C05454=1112.944,404.001,-92.503,-176.618,11.577,149.492
C05455=1112.941,404.248,-92.543,-176.616,11.582,149.493
C05456=1112.937,404.494,-92.582,-176.614,11.587,149.494
C05457=1112.933,404.741,-92.621,-176.613,11.591,149.494
C05458=1112.930,404.988,-92.660,-176.611,11.596,149.495
C05459=1112.927,405.235,-92.699,-176.609,11.601,149.496
C05460=1112.923,405.482,-92.738,-176.606,11.605,149.496
C05461=1112.920,405.729,-92.778,-176.604,11.610,149.497
C05462=1112.916,405.976,-92.817,-176.603,11.615,149.498
C05463=1112.913,406.223,-92.856,-176.601,11.620,149.499
C05464=1112.909,406.470,-92.895,-176.599,11.625,149.500
C05465=1112.905,406.717,-92.935,-176.597,11.630,149.501
C05466=1112.902,406.964,-92.974,-176.595,11.635,149.501
C05467=1112.898,407.211,-93.013,-176.593,11.640,149.502
C05468=1112.895,407.457,-93.052,-176.592,11.645,149.503
C05469=1112.892,407.704,-93.091,-176.590,11.650,149.504
C05470=1112.888,407.951,-93.131,-176.588,11.655,149.505
C05471=1112.885,408.198,-93.170,-176.586,11.660,149.506
C05472=1112.881,408.445,-93.209,-176.584,11.665,149.507
C05473=1112.877,408.692,-93.249,-176.583,11.671,149.508
C05474=1112.874,408.939,-93.288,-176.581,11.677,149.509
C05475=1112.870,409.186,-93.327,-176.579,11.681,149.509
C05476=1112.867,409.432,-93.367,-176.577,11.687,149.510
C05477=1112.863,409.679,-93.406,-176.576,11.692,149.511
C05478=1112.860,409.926,-93.446,-176.574,11.697,149.512
C05479=1112.856,410.173,-93.485,-176.572,11.703,149.513
C05480=1112.853,410.419,-93.525,-176.570,11.708,149.514
C05481=1112.849,410.666,-93.564,-176.569,11.714,149.516
C05482=1112.845,410.913,-93.603,-176.567,11.720,149.517
C05483=1112.842,411.160,-93.643,-176.565,11.725,149.518
C05484=1112.839,411.407,-93.683,-176.564,11.731,149.519
C05485=1112.835,411.654,-93.722,-176.562,11.737,149.520
C05486=1112.832,411.900,-93.762,-176.561,11.742,149.521
C05487=1112.829,412.147,-93.801,-176.558,11.748,149.522
C05488=1112.824,412.395,-93.841,-176.557,11.754,149.523
C05489=1112.821,412.641,-93.881,-176.555,11.760,149.524
C05490=1112.817,412.888,-93.920,-176.554,11.765,149.525
C05491=1112.814,413.134,-93.960,-176.552,11.772,149.526
C05492=1112.810,413.381,-94.000,-176.551,11.777,149.528
C05493=1112.808,413.628,-94.040,-176.549,11.784,149.529
C05494=1112.805,413.875,-94.079,-176.548,11.789,149.530
C05495=1112.802,414.122,-94.119,-176.546,11.795,149.531
C05496=1112.801,414.368,-94.158,-176.544,11.802,149.533
C05497=1112.799,414.616,-94.198,-176.543,11.808,149.534
C05498=1112.800,414.863,-94.237,-176.541,11.814,149.535
C05499=1112.799,415.110,-94.277,-176.541,11.820,149.536
C05500=1112.799,415.356,-94.316,-176.539,11.826,149.537
C05501=1112.800,415.603,-94.356,-176.537,11.833,149.539
C05502=1112.802,415.814,-94.389,-176.536,11.838,149.540
C05503=1112.802,416.025,-94.422,-176.535,11.843,149.541
C05504=1112.805,416.236,-94.456,-176.534,11.849,149.542
C05505=1112.807,416.448,-94.489,-176.533,11.854,149.543
C05506=1112.810,416.659,-94.522,-176.532,11.860,149.545
C05507=1112.813,416.870,-94.555,-176.531,11.865,149.546
C05508=1112.817,417.081,-94.589,-176.529,11.871,149.547
C05509=1112.820,417.292,-94.622,-176.528,11.877,149.548
C05510=1112.401,417.292,-94.684,-176.521,11.881,149.547
C05511=1112.398,417.081,-94.652,-176.522,11.875,149.546
C05512=1112.394,416.870,-94.618,-176.523,11.870,149.545
C05513=1112.391,416.659,-94.585,-176.524,11.864,149.544
C05514=1112.388,416.448,-94.552,-176.526,11.858,149.543
C05515=1112.386,416.236,-94.519,-176.527,11.853,149.541
C05516=1112.384,416.025,-94.485,-176.528,11.847,149.540
C05517=1112.383,415.814,-94.451,-176.529,11.842,149.539
C05518=1112.381,415.602,-94.417,-176.530,11.836,149.538
C05519=1112.380,415.356,-94.378,-176.532,11.831,149.537
C05520=1112.379,415.109,-94.339,-176.533,11.824,149.535
C05521=1112.380,414.862,-94.300,-176.535,11.818,149.534
C05522=1112.381,414.615,-94.260,-176.536,11.812,149.533
C05523=1112.382,414.368,-94.221,-176.538,11.806,149.532
C05524=1112.384,414.122,-94.181,-176.539,11.799,149.531
C05525=1112.386,413.875,-94.141,-176.541,11.794,149.529
C05526=1112.388,413.628,-94.102,-176.543,11.787,149.528
C05527=1112.391,413.381,-94.062,-176.544,11.781,149.527
C05528=1112.395,413.135,-94.022,-176.546,11.776,149.526
C05529=1112.398,412.888,-93.983,-176.547,11.769,149.525
C05530=1112.401,412.641,-93.943,-176.549,11.764,149.523
C05531=1112.405,412.393,-93.903,-176.551,11.758,149.522
C05532=1112.409,412.147,-93.863,-176.552,11.752,149.521
C05533=1112.412,411.900,-93.824,-176.554,11.746,149.520
C05534=1112.416,411.653,-93.785,-176.555,11.741,149.519
C05535=1112.419,411.407,-93.745,-176.558,11.735,149.518
C05536=1112.423,411.160,-93.705,-176.559,11.729,149.517
C05537=1112.426,410.913,-93.666,-176.561,11.723,149.516
C05538=1112.430,410.667,-93.626,-176.563,11.718,149.515
C05539=1112.433,410.420,-93.587,-176.565,11.712,149.514
C05540=1112.437,410.173,-93.548,-176.566,11.707,149.513
C05541=1112.440,409.926,-93.507,-176.568,11.701,149.512
C05542=1112.443,409.679,-93.468,-176.570,11.695,149.511
C05543=1112.447,409.432,-93.429,-176.572,11.690,149.510
C05544=1112.451,409.185,-93.390,-176.573,11.685,149.509
C05545=1112.454,408.938,-93.350,-176.575,11.680,149.508
C05546=1112.458,408.691,-93.310,-176.577,11.674,149.507
C05547=1112.461,408.445,-93.271,-176.579,11.669,149.506
C05548=1112.465,408.198,-93.232,-176.581,11.663,149.505
C05549=1112.468,407.951,-93.193,-176.583,11.659,149.504
C05550=1112.472,407.704,-93.153,-176.584,11.653,149.503
C05551=1112.475,407.457,-93.113,-176.586,11.648,149.503
C05552=1112.479,407.210,-93.074,-176.588,11.642,149.502
C05553=1112.483,406.963,-93.035,-176.590,11.638,149.501
C05554=1112.486,406.716,-92.996,-176.592,11.633,149.500
C05555=1112.490,406.469,-92.956,-176.594,11.628,149.499
C05556=1112.493,406.222,-92.917,-176.596,11.623,149.499
C05557=1112.496,405.976,-92.878,-176.598,11.618,149.498
C05558=1112.500,405.729,-92.839,-176.600,11.613,149.497
C05559=1112.504,405.482,-92.800,-176.602,11.608,149.496
C05560=1112.507,405.235,-92.761,-176.604,11.603,149.495
C05561=1112.511,404.988,-92.721,-176.606,11.598,149.495
C05562=1112.514,404.741,-92.682,-176.608,11.593,149.494
C05563=1112.518,404.494,-92.643,-176.609,11.589,149.493
C05564=1112.521,404.248,-92.605,-176.612,11.585,149.492
C05565=1112.525,404.001,-92.565,-176.614,11.580,149.492
C05566=1112.529,403.754,-92.526,-176.616,11.575,149.491
C05567=1112.532,403.543,-92.493,-176.618,11.571,149.490
C05568=1112.535,403.331,-92.459,-176.619,11.568,149.490
C05569=1112.538,403.120,-92.426,-176.621,11.564,149.489
C05570=1112.540,402.908,-92.393,-176.623,11.560,149.489
C05571=1112.544,402.697,-92.360,-176.625,11.555,149.488
C05572=1112.547,402.486,-92.326,-176.627,11.552,149.488
C05573=1112.550,402.274,-92.293,-176.629,11.548,149.487
C05574=1112.553,402.063,-92.259,-176.630,11.544,149.487
C05575=1112.556,401.816,-92.221,-176.632,11.540,149.486
C05576=1112.560,401.569,-92.181,-176.634,11.536,149.485
C05577=1112.563,401.322,-92.142,-176.637,11.531,149.485
C05578=1112.567,401.075,-92.104,-176.639,11.527,149.484
C05579=1112.571,400.829,-92.065,-176.641,11.523,149.484
C05580=1112.574,400.582,-92.026,-176.643,11.518,149.483
C05581=1112.578,400.334,-91.988,-176.645,11.514,149.482
C05582=1112.581,400.087,-91.949,-176.648,11.510,149.482
C05583=1112.585,399.841,-91.910,-176.649,11.506,149.481
C05584=1112.589,399.593,-91.871,-176.652,11.502,149.481
C05585=1112.592,399.347,-91.833,-176.654,11.498,149.480
C05586=1112.596,399.100,-91.794,-176.656,11.494,149.480
C05587=1112.600,398.852,-91.755,-176.658,11.490,149.479
C05588=1112.603,398.606,-91.716,-176.661,11.486,149.479
C05589=1112.606,398.359,-91.677,-176.663,11.482,149.479
C05590=1112.611,398.112,-91.639,-176.666,11.478,149.478
C05591=1112.614,397.865,-91.600,-176.667,11.474,149.478
C05592=1112.618,397.618,-91.562,-176.669,11.471,149.477
C05593=1112.621,397.371,-91.522,-176.672,11.466,149.477
C05594=1112.624,397.123,-91.485,-176.674,11.463,149.476
C05595=1112.629,396.877,-91.446,-176.676,11.459,149.476
C05596=1112.632,396.630,-91.408,-176.679,11.455,149.476
C05597=1112.636,396.383,-91.368,-176.681,11.452,149.475
C05598=1112.639,396.136,-91.331,-176.683,11.448,149.475
C05599=1112.643,395.889,-91.292,-176.686,11.444,149.474
C05600=1112.647,395.642,-91.253,-176.688,11.440,149.474
C05601=1112.650,395.395,-91.215,-176.690,11.437,149.474
C05602=1112.654,395.148,-91.176,-176.692,11.434,149.473
C05603=1112.657,394.901,-91.138,-176.695,11.430,149.473
C05604=1112.661,394.654,-91.099,-176.698,11.426,149.473
C05605=1112.664,394.407,-91.061,-176.700,11.423,149.472
C05606=1112.669,394.160,-91.023,-176.702,11.420,149.472
C05607=1112.672,393.913,-90.984,-176.704,11.416,149.472
C05608=1112.676,393.666,-90.946,-176.707,11.413,149.472
C05609=1112.679,393.419,-90.908,-176.709,11.409,149.471
C05610=1112.683,393.172,-90.869,-176.711,11.406,149.471
C05611=1112.686,392.925,-90.831,-176.714,11.402,149.471
C05612=1112.690,392.677,-90.792,-176.717,11.399,149.470
C05613=1112.694,392.431,-90.755,-176.719,11.396,149.470
C05614=1112.698,392.184,-90.716,-176.722,11.393,149.470
C05615=1112.701,391.937,-90.678,-176.724,11.389,149.470
C05616=1112.704,391.690,-90.640,-176.726,11.386,149.470
C05617=1112.708,391.442,-90.602,-176.729,11.383,149.469
C05618=1112.712,391.195,-90.564,-176.731,11.380,149.469
C05619=1112.716,390.949,-90.525,-176.734,11.377,149.469
C05620=1112.719,390.702,-90.487,-176.736,11.373,149.469
C05621=1112.722,390.454,-90.449,-176.738,11.371,149.469
C05622=1112.727,390.207,-90.411,-176.741,11.368,149.468
C05623=1112.729,389.996,-90.378,-176.743,11.365,149.468
C05624=1112.733,389.784,-90.346,-176.745,11.363,149.468
C05625=1112.736,389.573,-90.313,-176.747,11.360,149.468
C05626=1112.739,389.361,-90.280,-176.750,11.357,149.468
C05627=1112.742,389.150,-90.248,-176.752,11.355,149.468
C05628=1112.745,388.938,-90.215,-176.754,11.353,149.468
C05629=1112.748,388.726,-90.183,-176.756,11.350,149.468
C05630=1112.751,388.516,-90.151,-176.758,11.347,149.468
C05631=1112.755,388.268,-90.112,-176.761,11.344,149.468
C05632=1112.759,388.021,-90.074,-176.763,11.342,149.467
C05633=1112.762,387.774,-90.037,-176.766,11.339,149.467
C05634=1112.766,387.527,-89.998,-176.768,11.336,149.467
C05635=1112.770,387.280,-89.960,-176.771,11.333,149.467
C05636=1112.773,387.033,-89.922,-176.773,11.331,149.467
C05637=1112.777,386.786,-89.885,-176.776,11.328,149.467
C05638=1112.781,386.539,-89.846,-176.779,11.325,149.467
C05639=1112.784,386.291,-89.808,-176.781,11.323,149.467
C05640=1112.788,386.045,-89.771,-176.784,11.320,149.467
C05641=1112.791,385.797,-89.733,-176.787,11.317,149.467
C05642=1112.795,385.551,-89.695,-176.789,11.315,149.467
C05643=1112.799,385.303,-89.657,-176.791,11.312,149.467
C05644=1112.803,385.056,-89.620,-176.794,11.309,149.467
C05645=1112.806,384.809,-89.582,-176.797,11.307,149.467
C05646=1112.810,384.562,-89.544,-176.799,11.305,149.467
C05647=1112.813,384.315,-89.506,-176.802,11.302,149.467
C05648=1112.817,384.068,-89.468,-176.805,11.300,149.467
C05649=1112.821,383.820,-89.431,-176.807,11.298,149.467
C05650=1112.825,383.574,-89.394,-176.810,11.295,149.467
C05651=1112.828,383.326,-89.356,-176.813,11.292,149.467
C05652=1112.832,383.080,-89.317,-176.816,11.290,149.467
C05653=1112.836,382.832,-89.280,-176.819,11.287,149.468
C05654=1112.840,382.585,-89.243,-176.822,11.284,149.468
C05655=1112.843,382.338,-89.205,-176.825,11.282,149.468
C05656=1112.847,382.091,-89.167,-176.828,11.279,149.468
C05657=1112.850,381.843,-89.130,-176.832,11.276,149.468
C05658=1112.854,381.597,-89.092,-176.836,11.273,149.468
C05659=1112.857,381.349,-89.054,-176.838,11.270,149.468
C05660=1112.861,381.102,-89.017,-176.842,11.268,149.468
C05661=1112.865,380.855,-88.979,-176.845,11.265,149.468
C05662=1112.869,380.608,-88.942,-176.848,11.263,149.469
C05663=1112.873,380.361,-88.905,-176.851,11.260,149.469
C05664=1112.876,380.114,-88.867,-176.854,11.258,149.469
C05665=1112.880,379.866,-88.830,-176.858,11.255,149.469
C05666=1112.883,379.619,-88.792,-176.861,11.252,149.469
C05667=1112.887,379.372,-88.755,-176.864,11.250,149.469
C05668=1112.891,379.125,-88.717,-176.867,11.247,149.469
C05669=1112.895,378.878,-88.680,-176.871,11.245,149.470
C05670=1112.899,378.631,-88.643,-176.874,11.242,149.470
C05671=1112.902,378.383,-88.605,-176.877,11.239,149.470
C05672=1112.906,378.137,-88.568,-176.880,11.237,149.470
C05673=1112.910,377.889,-88.531,-176.884,11.234,149.470
C05674=1112.913,377.642,-88.493,-176.887,11.231,149.470
C05675=1112.917,377.395,-88.456,-176.891,11.229,149.471
C05676=1112.921,377.148,-88.419,-176.894,11.226,149.471
C05677=1112.924,376.900,-88.381,-176.897,11.224,149.471
C05678=1112.929,376.653,-88.344,-176.900,11.221,149.471
C05679=1112.931,376.441,-88.312,-176.903,11.219,149.471
C05680=1112.935,376.230,-88.281,-176.906,11.217,149.472
C05681=1112.938,376.019,-88.249,-176.908,11.215,149.472
C05682=1112.941,375.807,-88.217,-176.911,11.213,149.472
C05683=1112.944,375.595,-88.186,-176.914,11.211,149.472
C05684=1112.947,375.383,-88.154,-176.917,11.209,149.472
C05685=1112.951,375.172,-88.121,-176.920,11.206,149.472
C05686=1112.954,374.960,-88.089,-176.922,11.204,149.473
C05687=1112.958,374.712,-88.053,-176.926,11.202,149.473
C05688=1112.961,374.465,-88.016,-176.929,11.199,149.473
C05689=1112.965,374.218,-87.979,-176.932,11.197,149.473
C05690=1112.969,373.970,-87.942,-176.936,11.194,149.473
C05691=1112.972,373.724,-87.905,-176.939,11.192,149.474
C05692=1112.977,373.477,-87.868,-176.942,11.190,149.474
C05693=1112.979,373.229,-87.831,-176.946,11.187,149.474
C05694=1112.983,372.982,-87.794,-176.949,11.185,149.474
C05695=1112.987,372.735,-87.757,-176.952,11.182,149.474
C05696=1112.992,372.487,-87.721,-176.955,11.180,149.475
C05697=1112.995,372.240,-87.683,-176.959,11.177,149.475
C05698=1112.998,371.993,-87.646,-176.962,11.175,149.475
C05699=1113.002,371.746,-87.609,-176.965,11.172,149.475
C05700=1113.006,371.499,-87.573,-176.969,11.170,149.475
C05701=1113.010,371.251,-87.535,-176.972,11.167,149.476
C05702=1113.013,371.004,-87.499,-176.975,11.165,149.476
C05703=1113.017,370.757,-87.462,-176.979,11.163,149.476
C05704=1113.021,370.510,-87.425,-176.982,11.160,149.476
C05705=1113.025,370.263,-87.389,-176.986,11.158,149.477
C05706=1113.028,370.015,-87.352,-176.989,11.155,149.477
C05707=1113.032,369.768,-87.315,-176.992,11.153,149.477
C05708=1113.036,369.521,-87.278,-176.995,11.150,149.477
C05709=1113.040,369.274,-87.242,-176.999,11.148,149.477
C05710=1113.044,369.026,-87.206,-177.002,11.145,149.478
C05711=1113.047,368.778,-87.169,-177.006,11.143,149.478
C05712=1113.051,368.531,-87.132,-177.009,11.141,149.478
C05713=1113.055,368.284,-87.095,-177.012,11.138,149.478
C05714=1113.058,368.037,-87.059,-177.016,11.136,149.479
C05715=1113.063,367.790,-87.022,-177.019,11.133,149.479
C05716=1113.067,367.543,-86.985,-177.022,11.131,149.479
C05717=1113.070,367.295,-86.950,-177.026,11.129,149.479
C05718=1113.074,367.047,-86.913,-177.029,11.126,149.480
C05719=1113.077,366.800,-86.876,-177.033,11.124,149.480
C05720=1113.081,366.553,-86.840,-177.036,11.121,149.480
C05721=1113.086,366.305,-86.803,-177.039,11.119,149.480
C05722=1113.089,366.059,-86.767,-177.043,11.116,149.481
C05723=1113.093,365.811,-86.730,-177.046,11.114,149.481
C05724=1113.096,365.565,-86.694,-177.049,11.112,149.481
C05725=1113.101,365.317,-86.658,-177.053,11.109,149.481
C05726=1113.104,365.069,-86.621,-177.056,11.107,149.482
C05727=1113.108,364.822,-86.584,-177.060,11.104,149.482
C05728=1113.111,364.574,-86.549,-177.063,11.102,149.482
C05729=1113.115,364.327,-86.512,-177.066,11.099,149.482
C05730=1113.119,364.080,-86.476,-177.070,11.097,149.483
C05731=1113.123,363.833,-86.440,-177.073,11.095,149.483
C05732=1113.127,363.586,-86.403,-177.077,11.092,149.483
C05733=1113.131,363.338,-86.367,-177.080,11.090,149.483
C05734=1113.134,363.091,-86.331,-177.083,11.088,149.484
C05735=1113.138,362.879,-86.300,-177.086,11.086,149.484
C05736=1113.140,362.667,-86.269,-177.089,11.084,149.484
C05737=1113.144,362.455,-86.238,-177.092,11.082,149.484
C05738=1113.147,362.243,-86.207,-177.095,11.080,149.485
C05739=1113.150,362.032,-86.177,-177.097,11.078,149.485
C05740=1113.154,361.820,-86.146,-177.100,11.075,149.485
C05741=1113.157,361.607,-86.114,-177.103,11.074,149.485
C05742=1113.159,361.396,-86.083,-177.106,11.071,149.485
C05743=1113.164,361.148,-86.047,-177.109,11.069,149.486
C05744=1113.168,360.901,-86.012,-177.113,11.067,149.486
C05745=1113.172,360.654,-85.975,-177.116,11.064,149.486
C05746=1113.175,360.406,-85.939,-177.120,11.062,149.486
C05747=1113.179,360.159,-85.903,-177.123,11.059,149.487
C05748=1113.183,359.912,-85.867,-177.126,11.057,149.487
C05749=1113.187,359.664,-85.831,-177.130,11.055,149.487
C05750=1113.190,359.417,-85.795,-177.133,11.052,149.487
C05751=1113.194,359.170,-85.759,-177.137,11.050,149.488
C05752=1113.198,358.922,-85.723,-177.140,11.047,149.488
C05753=1113.201,358.675,-85.687,-177.143,11.045,149.488
C05754=1113.205,358.427,-85.651,-177.147,11.043,149.488
C05755=1113.209,358.180,-85.616,-177.150,11.040,149.489
C05756=1113.213,357.932,-85.580,-177.154,11.038,149.489
C05757=1113.217,357.686,-85.544,-177.157,11.035,149.489
C05758=1113.221,357.438,-85.508,-177.160,11.034,149.489
C05759=1113.224,357.191,-85.473,-177.163,11.031,149.490
C05760=1113.229,356.943,-85.437,-177.167,11.029,149.490
C05761=1113.233,356.696,-85.401,-177.170,11.026,149.490
C05762=1113.236,356.449,-85.365,-177.174,11.023,149.490
C05763=1113.240,356.201,-85.329,-177.177,11.021,149.491
C05764=1113.243,355.954,-85.294,-177.180,11.018,149.491
C05765=1113.248,355.706,-85.258,-177.184,11.016,149.491
C05766=1113.251,355.458,-85.222,-177.187,11.014,149.491
C05767=1113.255,355.211,-85.187,-177.191,11.011,149.492
C05768=1113.259,354.964,-85.151,-177.194,11.009,149.492
C05769=1113.263,354.717,-85.116,-177.197,11.006,149.492
C05770=1113.267,354.469,-85.080,-177.201,11.004,149.492
C05771=1113.270,354.222,-85.045,-177.204,11.001,149.493
C05772=1113.275,353.974,-85.009,-177.207,10.999,149.493
C05773=1113.278,353.726,-84.973,-177.211,10.997,149.493
C05774=1113.282,353.479,-84.937,-177.214,10.994,149.493
C05775=1113.286,353.232,-84.902,-177.218,10.992,149.494
C05776=1113.290,352.985,-84.867,-177.221,10.989,149.494
C05777=1113.294,352.737,-84.831,-177.224,10.987,149.494
C05778=1113.297,352.490,-84.796,-177.228,10.984,149.494
C05779=1113.301,352.242,-84.760,-177.231,10.982,149.495
C05780=1113.305,351.995,-84.725,-177.234,10.980,149.495
C05781=1113.309,351.748,-84.689,-177.237,10.977,149.495
C05782=1113.313,351.500,-84.655,-177.241,10.975,149.495
C05783=1113.316,351.252,-84.619,-177.244,10.972,149.495
C05784=1113.320,351.005,-84.583,-177.247,10.970,149.496
C05785=1113.324,350.758,-84.548,-177.251,10.967,149.496
C05786=1113.328,350.510,-84.513,-177.254,10.965,149.496
C05787=1113.332,350.263,-84.477,-177.257,10.962,149.496
C05788=1113.336,350.015,-84.442,-177.261,10.960,149.497
C05789=1113.340,349.768,-84.407,-177.264,10.957,149.497
C05790=1113.344,349.520,-84.372,-177.268,10.954,149.497
C05791=1113.347,349.308,-84.342,-177.271,10.952,149.497
C05792=1113.350,349.096,-84.311,-177.273,10.951,149.498
C05793=1113.354,348.884,-84.281,-177.276,10.948,149.498
C05794=1113.357,348.672,-84.251,-177.279,10.946,149.498
C05795=1113.360,348.460,-84.221,-177.281,10.944,149.498
C05796=1113.363,348.248,-84.191,-177.284,10.942,149.498
C05797=1113.367,348.036,-84.161,-177.287,10.940,149.498
C05798=1113.370,347.824,-84.130,-177.289,10.938,149.498
C05799=1113.375,347.577,-84.096,-177.293,10.936,149.499
C05800=1113.378,347.329,-84.061,-177.296,10.933,149.499
C05801=1113.381,347.082,-84.025,-177.299,10.931,149.499
C05802=1113.386,346.834,-83.991,-177.302,10.928,149.499
C05803=1113.390,346.587,-83.955,-177.306,10.925,149.499
C05804=1113.394,346.339,-83.920,-177.309,10.923,149.500
C05805=1113.398,346.092,-83.885,-177.312,10.921,149.500
C05806=1113.402,345.844,-83.850,-177.316,10.918,149.500
C05807=1113.405,345.597,-83.815,-177.318,10.915,149.500
C05808=1113.409,345.349,-83.781,-177.321,10.914,149.500
C05809=1113.413,345.102,-83.745,-177.324,10.911,149.501
C05810=1113.417,344.854,-83.711,-177.328,10.909,149.501
C05811=1113.421,344.607,-83.675,-177.331,10.906,149.501
C05812=1113.424,344.359,-83.641,-177.334,10.904,149.501
C05813=1113.428,344.112,-83.606,-177.337,10.901,149.501
C05814=1113.433,343.864,-83.571,-177.341,10.899,149.502
C05815=1113.437,343.616,-83.536,-177.344,10.896,149.502
C05816=1113.441,343.369,-83.501,-177.347,10.894,149.502
C05817=1113.444,343.121,-83.467,-177.351,10.891,149.502
C05818=1113.448,342.873,-83.432,-177.353,10.888,149.502
C05819=1113.452,342.626,-83.397,-177.356,10.887,149.503
C05820=1113.456,342.379,-83.363,-177.359,10.884,149.503
C05821=1113.460,342.131,-83.328,-177.363,10.882,149.503
C05822=1113.464,341.884,-83.293,-177.366,10.879,149.503
C05823=1113.468,341.636,-83.258,-177.369,10.877,149.503
C05824=1113.472,341.389,-83.224,-177.372,10.874,149.504
C05825=1113.476,341.140,-83.189,-177.376,10.872,149.504
C05826=1113.480,340.894,-83.154,-177.379,10.869,149.504
C05827=1113.483,340.646,-83.120,-177.382,10.866,149.504
C05828=1113.488,340.398,-83.085,-177.385,10.864,149.504
C05829=1113.492,340.150,-83.050,-177.388,10.862,149.505
C05830=1113.495,339.903,-83.016,-177.391,10.860,149.505
C05831=1113.499,339.656,-82.981,-177.394,10.857,149.505
C05832=1113.503,339.409,-82.947,-177.397,10.855,149.505
C05833=1113.507,339.160,-82.912,-177.401,10.852,149.505
C05834=1113.511,338.913,-82.878,-177.404,10.850,149.506
C05835=1113.515,338.665,-82.843,-177.407,10.847,149.506
C05836=1113.519,338.418,-82.809,-177.410,10.844,149.506
C05837=1113.523,338.170,-82.775,-177.414,10.842,149.506
C05838=1113.527,337.923,-82.740,-177.417,10.840,149.506
C05839=1113.531,337.674,-82.705,-177.420,10.837,149.507
C05840=1113.535,337.427,-82.672,-177.423,10.835,149.507
C05841=1113.539,337.179,-82.637,-177.426,10.833,149.507
C05842=1113.543,336.932,-82.603,-177.429,10.830,149.507
C05843=1113.547,336.684,-82.568,-177.432,10.828,149.507
C05844=1113.550,336.437,-82.534,-177.435,10.825,149.507
C05845=1113.555,336.189,-82.500,-177.439,10.822,149.508
C05846=1113.558,335.942,-82.465,-177.442,10.820,149.508
C05847=1113.562,335.729,-82.436,-177.444,10.818,149.508
C05848=1113.565,335.518,-82.407,-177.448,10.816,149.508
C05849=1113.569,335.306,-82.377,-177.450,10.814,149.508
C05850=1113.572,335.093,-82.347,-177.453,10.812,149.509
C05851=1113.575,334.880,-82.319,-177.456,10.809,149.509
C05852=1113.579,334.669,-82.289,-177.458,10.807,149.509
C05853=1113.582,334.457,-82.260,-177.460,10.805,149.509
C05854=1113.585,334.245,-82.231,-177.464,10.803,149.509
C05855=1113.589,333.997,-82.196,-177.467,10.800,149.509
C05856=1113.593,333.749,-82.163,-177.470,10.798,149.509
C05857=1113.597,333.501,-82.128,-177.473,10.796,149.510
C05858=1113.601,333.254,-82.094,-177.476,10.794,149.510
C05859=1113.605,333.006,-82.060,-177.479,10.791,149.510
C05860=1113.609,332.759,-82.026,-177.482,10.788,149.510
C05861=1113.613,332.511,-81.993,-177.486,10.786,149.511
C05862=1113.616,332.264,-81.958,-177.489,10.783,149.511
C05863=1113.621,332.016,-81.924,-177.492,10.781,149.511
C05864=1113.625,331.768,-81.890,-177.495,10.778,149.511
C05865=1113.628,331.521,-81.856,-177.498,10.776,149.511
C05866=1113.633,331.273,-81.822,-177.501,10.773,149.511
C05867=1113.637,331.025,-81.788,-177.505,10.771,149.512
C05868=1113.640,330.778,-81.755,-177.507,10.769,149.512
C05869=1113.645,330.530,-81.720,-177.510,10.766,149.512
C05870=1113.648,330.282,-81.687,-177.514,10.764,149.512
C05871=1113.652,330.035,-81.653,-177.517,10.761,149.512
C05872=1113.656,329.788,-81.619,-177.520,10.758,149.512
C05873=1113.660,329.539,-81.585,-177.523,10.756,149.513
C05874=1113.664,329.292,-81.551,-177.527,10.754,149.513
C05875=1113.668,329.044,-81.518,-177.530,10.751,149.513
C05876=1113.672,328.797,-81.484,-177.533,10.748,149.513
C05877=1113.676,328.548,-81.450,-177.536,10.746,149.514
C05878=1113.680,328.301,-81.416,-177.539,10.743,149.514
C05879=1113.684,328.053,-81.383,-177.542,10.741,149.514
C05880=1113.688,327.805,-81.348,-177.545,10.739,149.514
C05881=1113.692,327.558,-81.315,-177.548,10.736,149.514
C05882=1113.696,327.310,-81.281,-177.551,10.734,149.514
C05883=1113.700,327.063,-81.248,-177.555,10.731,149.515
C05884=1113.704,326.815,-81.213,-177.558,10.729,149.515
C05885=1113.708,326.567,-81.180,-177.561,10.726,149.515
C05886=1113.712,326.319,-81.147,-177.564,10.724,149.515
C05887=1113.716,326.072,-81.113,-177.567,10.721,149.515
C05888=1113.719,325.824,-81.080,-177.570,10.718,149.515
C05889=1113.724,325.576,-81.047,-177.574,10.716,149.516
C05890=1113.728,325.329,-81.012,-177.576,10.714,149.516
C05891=1113.732,325.081,-80.979,-177.579,10.711,149.516
C05892=1113.736,324.833,-80.946,-177.583,10.709,149.516
C05893=1113.740,324.585,-80.912,-177.586,10.707,149.517
C05894=1113.744,324.338,-80.878,-177.589,10.704,149.517
C05895=1113.748,324.090,-80.845,-177.592,10.701,149.517
C05896=1113.752,323.843,-80.811,-177.596,10.699,149.517
C05897=1113.756,323.595,-80.778,-177.598,10.696,149.517
C05898=1113.759,323.347,-80.745,-177.602,10.694,149.517
C05899=1113.764,323.099,-80.712,-177.605,10.691,149.517
C05900=1113.768,322.851,-80.678,-177.608,10.688,149.518
C05901=1113.771,322.604,-80.645,-177.611,10.687,149.518
C05902=1113.776,322.356,-80.611,-177.614,10.684,149.518
C05903=1113.779,322.143,-80.582,-177.617,10.682,149.518
C05904=1113.783,321.932,-80.555,-177.619,10.680,149.518
C05905=1113.786,321.719,-80.526,-177.622,10.678,149.519
C05906=1113.789,321.507,-80.498,-177.625,10.675,149.519
C05907=1113.793,321.295,-80.468,-177.627,10.673,149.519
C05908=1113.796,321.083,-80.440,-177.630,10.671,149.519
C05909=1113.800,320.870,-80.411,-177.633,10.669,149.519
C05910=1113.803,320.658,-80.383,-177.636,10.667,149.519
C05911=1113.806,320.410,-80.350,-177.638,10.664,149.520
C05912=1113.811,320.162,-80.317,-177.642,10.662,149.520
C05913=1113.815,319.914,-80.284,-177.645,10.659,149.520
C05914=1113.819,319.666,-80.250,-177.648,10.657,149.520
C05915=1113.822,319.419,-80.218,-177.651,10.654,149.520
C05916=1113.826,319.171,-80.185,-177.654,10.651,149.520
C05917=1113.831,318.924,-80.152,-177.657,10.650,149.521
C05918=1113.835,318.676,-80.118,-177.660,10.647,149.521
C05919=1113.839,318.428,-80.085,-177.663,10.644,149.521
C05920=1113.843,318.180,-80.052,-177.667,10.642,149.521
C05921=1113.847,317.933,-80.019,-177.669,10.639,149.521
C05922=1113.850,317.685,-79.986,-177.673,10.637,149.522
C05923=1113.854,317.437,-79.953,-177.676,10.634,149.522
C05924=1113.858,317.188,-79.920,-177.679,10.632,149.522
C05925=1113.863,316.941,-79.887,-177.682,10.629,149.522
C05926=1113.867,316.693,-79.854,-177.685,10.626,149.522
C05927=1113.870,316.446,-79.822,-177.689,10.624,149.522
C05928=1113.874,316.198,-79.788,-177.691,10.622,149.523
C05929=1113.878,315.950,-79.755,-177.694,10.619,149.523
C05930=1113.883,315.702,-79.723,-177.698,10.617,149.523
C05931=1113.886,315.454,-79.690,-177.700,10.614,149.523
C05932=1113.890,315.207,-79.657,-177.704,10.612,149.523
C05933=1113.895,314.959,-79.624,-177.707,10.609,149.523
C05934=1113.899,314.711,-79.591,-177.710,10.607,149.524
C05935=1113.902,314.463,-79.559,-177.713,10.604,149.524
C05936=1113.907,314.215,-79.526,-177.716,10.601,149.524
C05937=1113.911,313.968,-79.493,-177.720,10.599,149.524
C05938=1113.914,313.720,-79.461,-177.722,10.597,149.524
C05939=1113.919,313.472,-79.428,-177.725,10.595,149.525
C05940=1113.923,313.224,-79.394,-177.729,10.592,149.525
C05941=1113.926,312.976,-79.363,-177.732,10.589,149.525
C05942=1113.931,312.728,-79.329,-177.735,10.587,149.525
C05943=1113.935,312.480,-79.297,-177.738,10.584,149.525
C05944=1113.938,312.233,-79.264,-177.741,10.582,149.526
C05945=1113.943,311.986,-79.232,-177.744,10.579,149.526
C05946=1113.948,311.737,-79.199,-177.747,10.576,149.526
C05947=1113.951,311.490,-79.167,-177.751,10.574,149.526
C05948=1113.955,311.241,-79.134,-177.754,10.571,149.526
C05949=1113.959,310.994,-79.102,-177.756,10.570,149.527
C05950=1113.963,310.746,-79.069,-177.759,10.567,149.527
C05951=1113.967,310.498,-79.036,-177.763,10.564,149.527
C05952=1113.971,310.250,-79.004,-177.765,10.562,149.527
C05953=1113.975,310.002,-78.971,-177.769,10.559,149.527
C05954=1113.979,309.754,-78.939,-177.772,10.556,149.527
C05955=1113.983,309.506,-78.906,-177.775,10.554,149.528
C05956=1113.987,309.259,-78.875,-177.778,10.552,149.528
C05957=1113.992,309.011,-78.842,-177.781,10.549,149.528
C05958=1113.996,308.763,-78.809,-177.785,10.546,149.528
C05959=1114.000,308.551,-78.782,-177.787,10.544,149.528
C05960=1114.002,308.338,-78.754,-177.789,10.542,149.528
C05961=1114.006,308.125,-78.726,-177.793,10.540,149.529
C05962=1114.009,307.914,-78.698,-177.795,10.538,149.529
C05963=1114.013,307.700,-78.671,-177.797,10.536,149.529
C05964=1114.016,307.489,-78.643,-177.801,10.533,149.529
C05965=1114.020,307.276,-78.616,-177.803,10.531,149.529
C05966=1114.024,307.063,-78.588,-177.805,10.529,149.529
C05967=1114.027,306.816,-78.555,-177.808,10.527,149.529
C05968=1114.031,306.568,-78.523,-177.811,10.524,149.530
C05969=1114.036,306.319,-78.491,-177.815,10.522,149.530
C05970=1114.039,306.071,-78.459,-177.818,10.519,149.530
C05971=1114.044,305.824,-78.426,-177.821,10.517,149.530
C05972=1114.048,305.576,-78.395,-177.824,10.514,149.530
C05973=1114.052,305.328,-78.362,-177.827,10.511,149.531
C05974=1114.056,305.080,-78.330,-177.830,10.510,149.531
C05975=1114.060,304.833,-78.299,-177.833,10.507,149.531
C05976=1114.064,304.585,-78.266,-177.836,10.505,149.531
C05977=1114.068,304.337,-78.234,-177.839,10.502,149.531
C05978=1114.072,304.089,-78.202,-177.842,10.499,149.531
C05979=1114.077,303.841,-78.170,-177.845,10.497,149.532
C05980=1114.081,303.593,-78.138,-177.849,10.494,149.532
C05981=1114.085,303.345,-78.106,-177.852,10.491,149.532
C05982=1114.089,303.097,-78.074,-177.855,10.489,149.532
C05983=1114.093,302.849,-78.042,-177.858,10.486,149.532
C05984=1114.097,302.601,-78.010,-177.861,10.485,149.533
C05985=1114.101,302.353,-77.978,-177.864,10.482,149.533
C05986=1114.105,302.105,-77.946,-177.867,10.479,149.533
C05987=1114.109,301.858,-77.915,-177.870,10.477,149.533
C05988=1114.114,301.609,-77.882,-177.873,10.474,149.533
C05989=1114.117,301.361,-77.850,-177.876,10.471,149.533
C05990=1114.122,301.114,-77.819,-177.879,10.469,149.534
C05991=1114.126,300.866,-77.786,-177.882,10.466,149.534
C05992=1114.130,300.618,-77.755,-177.886,10.464,149.534
C05993=1114.134,300.370,-77.723,-177.889,10.461,149.534
C05994=1114.138,300.122,-77.691,-177.891,10.459,149.534
C05995=1114.141,299.874,-77.659,-177.894,10.457,149.534
C05996=1114.147,299.627,-77.627,-177.898,10.454,149.535
C05997=1114.150,299.378,-77.595,-177.900,10.451,149.535
C05998=1114.154,299.130,-77.564,-177.904,10.449,149.535
C05999=1114.159,298.882,-77.533,-177.907,10.446,149.535
C06000=1114.162,298.634,-77.501,-177.910,10.444,149.535
C06001=1114.167,298.386,-77.469,-177.913,10.441,149.535
C06002=1114.171,298.139,-77.437,-177.916,10.439,149.536
C06003=1114.175,297.890,-77.406,-177.919,10.436,149.536
C06004=1114.179,297.643,-77.375,-177.922,10.434,149.536
C06005=1114.183,297.395,-77.343,-177.925,10.431,149.536
C06006=1114.187,297.147,-77.311,-177.928,10.429,149.536
C06007=1114.191,296.899,-77.280,-177.931,10.426,149.536
C06008=1114.195,296.651,-77.248,-177.935,10.424,149.537
C06009=1114.199,296.403,-77.217,-177.937,10.421,149.537
C06010=1114.204,296.155,-77.184,-177.941,10.419,149.537
C06011=1114.208,295.906,-77.153,-177.944,10.416,149.537
C06012=1114.212,295.659,-77.122,-177.947,10.413,149.537
C06013=1114.216,295.411,-77.090,-177.949,10.411,149.538
C06014=1114.220,295.163,-77.059,-177.952,10.409,149.538
C06015=1114.223,294.951,-77.032,-177.956,10.406,149.538
C06016=1114.226,294.738,-77.005,-177.958,10.404,149.538
C06017=1114.230,294.525,-76.978,-177.960,10.402,149.538
C06018=1114.234,294.312,-76.951,-177.963,10.399,149.538
C06019=1114.237,294.100,-76.925,-177.966,10.398,149.539
C06020=1114.241,293.887,-76.897,-177.968,10.396,149.539
C06021=1114.244,293.675,-76.870,-177.971,10.393,149.539
C06022=1114.248,293.462,-76.844,-177.974,10.391,149.539
C06023=1114.252,293.215,-76.813,-177.977,10.389,149.539
C06024=1114.256,292.966,-76.782,-177.980,10.386,149.539
C06025=1114.260,292.719,-76.750,-177.983,10.383,149.539
C06026=1114.264,292.470,-76.719,-177.986,10.381,149.540
C06027=1114.268,292.222,-76.687,-177.989,10.378,149.540
C06028=1114.273,291.974,-76.656,-177.992,10.376,149.540
C06029=1114.276,291.726,-76.625,-177.995,10.374,149.540
C06030=1114.281,291.478,-76.594,-177.998,10.371,149.540
C06031=1114.285,291.229,-76.563,-178.001,10.369,149.541
C06032=1114.289,290.982,-76.531,-178.004,10.366,149.541
C06033=1114.294,290.734,-76.500,-178.007,10.363,149.541
C06034=1114.297,290.486,-76.469,-178.010,10.361,149.541
C06035=1114.302,290.238,-76.438,-178.013,10.358,149.541
C06036=1114.306,289.990,-76.407,-178.017,10.355,149.541
C06037=1114.310,289.742,-76.376,-178.019,10.353,149.541
C06038=1114.314,289.494,-76.345,-178.022,10.351,149.542
C06039=1114.318,289.246,-76.314,-178.025,10.348,149.542
C06040=1114.321,288.998,-76.283,-178.029,10.346,149.542
C06041=1114.326,288.750,-76.252,-178.032,10.343,149.542
C06042=1114.330,288.502,-76.221,-178.035,10.341,149.542
C06043=1114.335,288.254,-76.190,-178.038,10.338,149.543
C06044=1114.339,288.006,-76.159,-178.041,10.335,149.543
C06045=1114.342,287.758,-76.128,-178.044,10.333,149.543
C06046=1114.347,287.510,-76.097,-178.046,10.331,149.543
C06047=1114.351,287.261,-76.066,-178.050,10.328,149.543
C06048=1114.356,287.013,-76.035,-178.053,10.326,149.543
C06049=1114.359,286.766,-76.005,-178.056,10.323,149.544
C06050=1114.363,286.518,-75.973,-178.059,10.320,149.544
C06051=1114.368,286.270,-75.943,-178.062,10.318,149.544
C06052=1114.372,286.022,-75.912,-178.065,10.315,149.544
C06053=1114.376,285.773,-75.881,-178.068,10.312,149.544
C06054=1114.380,285.525,-75.851,-178.071,10.311,149.545
C06055=1114.384,285.277,-75.819,-178.074,10.308,149.545
C06056=1114.388,285.029,-75.789,-178.077,10.306,149.545
C06057=1114.393,284.781,-75.758,-178.080,10.303,149.545
C06058=1114.397,284.532,-75.727,-178.083,10.300,149.545
C06059=1114.401,284.285,-75.697,-178.086,10.298,149.545
C06060=1114.405,284.037,-75.666,-178.089,10.295,149.545
C06061=1114.409,283.788,-75.635,-178.093,10.292,149.546
C06062=1114.413,283.541,-75.605,-178.096,10.290,149.546
C06063=1114.418,283.293,-75.574,-178.098,10.288,149.546
C06064=1114.422,283.044,-75.543,-178.101,10.285,149.546
C06065=1114.426,282.796,-75.513,-178.104,10.282,149.546
C06066=1114.430,282.548,-75.482,-178.107,10.280,149.547
C06067=1114.434,282.301,-75.452,-178.110,10.277,149.547
C06068=1114.438,282.052,-75.421,-178.114,10.275,149.547
C06069=1114.443,281.804,-75.390,-178.117,10.272,149.547
C06070=1114.447,281.556,-75.360,-178.120,10.269,149.547
C06071=1114.450,281.344,-75.334,-178.122,10.268,149.547
C06072=1114.454,281.131,-75.308,-178.125,10.265,149.548
C06073=1114.457,280.918,-75.282,-178.128,10.263,149.548
C06074=1114.461,280.705,-75.255,-178.130,10.261,149.548
C06075=1114.465,280.493,-75.230,-178.133,10.259,149.548
C06076=1114.468,280.280,-75.204,-178.136,10.257,149.548
C06077=1114.472,280.067,-75.177,-178.138,10.254,149.548
C06078=1114.475,279.854,-75.151,-178.141,10.252,149.548
C06079=1114.479,279.606,-75.121,-178.144,10.249,149.549
C06080=1114.484,279.358,-75.091,-178.147,10.247,149.549
C06081=1114.488,279.110,-75.061,-178.150,10.244,149.549
C06082=1114.492,278.861,-75.030,-178.153,10.242,149.549
C06083=1114.496,278.614,-75.000,-178.156,10.239,149.549
C06084=1114.501,278.366,-74.969,-178.160,10.236,149.550
C06085=1114.505,278.117,-74.940,-178.163,10.234,149.550
C06086=1114.508,277.869,-74.909,-178.165,10.231,149.550
C06087=1114.513,277.621,-74.878,-178.168,10.228,149.550
C06088=1114.517,277.373,-74.849,-178.172,10.226,149.550
C06089=1114.521,277.125,-74.818,-178.175,10.223,149.550
C06090=1114.526,276.877,-74.789,-178.178,10.220,149.550
C06091=1114.530,276.629,-74.758,-178.181,10.217,149.550
C06092=1114.534,276.380,-74.727,-178.184,10.215,149.551
C06093=1114.538,276.132,-74.698,-178.187,10.212,149.551
C06094=1114.542,275.884,-74.668,-178.190,10.209,149.551
C06095=1114.547,275.636,-74.638,-178.193,10.207,149.551
C06096=1114.550,275.388,-74.607,-178.196,10.204,149.551
C06097=1114.555,275.140,-74.578,-178.199,10.201,149.551
C06098=1114.559,274.892,-74.547,-178.202,10.199,149.551
C06099=1114.563,274.643,-74.517,-178.204,10.197,149.552
C06100=1114.567,274.395,-74.487,-178.207,10.194,149.552
C06101=1114.572,274.147,-74.457,-178.210,10.191,149.552
C06102=1114.575,273.899,-74.427,-178.213,10.188,149.552
C06103=1114.580,273.651,-74.398,-178.216,10.186,149.552
C06104=1114.584,273.403,-74.368,-178.219,10.183,149.552
C06105=1114.588,273.155,-74.337,-178.222,10.180,149.552
C06106=1114.593,272.906,-74.308,-178.225,10.178,149.552
C06107=1114.596,272.659,-74.278,-178.228,10.175,149.553
C06108=1114.600,272.410,-74.248,-178.230,10.173,149.553
C06109=1114.605,272.161,-74.218,-178.233,10.170,149.553
C06110=1114.609,271.914,-74.188,-178.236,10.167,149.553
C06111=1114.613,271.665,-74.158,-178.239,10.165,149.553
C06112=1114.617,271.417,-74.129,-178.242,10.162,149.553
C06113=1114.621,271.169,-74.099,-178.245,10.159,149.553
C06114=1114.626,270.921,-74.069,-178.247,10.157,149.553
C06115=1114.630,270.673,-74.039,-178.250,10.154,149.553
C06116=1114.634,270.424,-74.010,-178.253,10.152,149.553
C06117=1114.639,270.176,-73.980,-178.256,10.149,149.554
C06118=1114.642,269.928,-73.950,-178.259,10.146,149.554
C06119=1114.647,269.680,-73.921,-178.261,10.144,149.554
C06120=1114.652,269.431,-73.891,-178.264,10.141,149.554
C06121=1114.656,269.183,-73.861,-178.267,10.139,149.554
C06122=1114.660,268.935,-73.832,-178.270,10.136,149.554
C06123=1114.664,268.687,-73.801,-178.273,10.133,149.554
C06124=1114.668,268.439,-73.772,-178.276,10.131,149.554
C06125=1114.672,268.191,-73.743,-178.278,10.128,149.554
C06126=1114.676,267.943,-73.713,-178.281,10.126,149.555
C06127=1114.680,267.729,-73.688,-178.284,10.124,149.555
C06128=1114.684,267.517,-73.662,-178.286,10.122,149.555
C06129=1114.687,267.304,-73.637,-178.288,10.120,149.555
C06130=1114.691,267.092,-73.612,-178.291,10.118,149.555
C06131=1114.695,266.878,-73.586,-178.294,10.115,149.555
C06132=1114.698,266.665,-73.561,-178.296,10.113,149.555
C06133=1114.702,266.453,-73.536,-178.298,10.111,149.555
C06134=1114.706,266.239,-73.511,-178.300,10.109,149.555
C06135=1114.710,265.991,-73.481,-178.303,10.106,149.555
C06136=1114.714,265.743,-73.452,-178.305,10.104,149.556
C06137=1114.718,265.494,-73.422,-178.308,10.101,149.556
C06138=1114.722,265.246,-73.393,-178.311,10.098,149.556
C06139=1114.727,264.999,-73.364,-178.314,10.096,149.556
C06140=1114.731,264.750,-73.334,-178.316,10.094,149.556
C06141=1114.736,264.502,-73.305,-178.320,10.091,149.556
C06142=1114.740,264.254,-73.275,-178.323,10.088,149.556
C06143=1114.744,264.005,-73.246,-178.326,10.086,149.556
C06144=1114.748,263.757,-73.216,-178.329,10.083,149.557
C06145=1114.752,263.509,-73.187,-178.332,10.081,149.557
C06146=1114.756,263.261,-73.158,-178.335,10.078,149.557
C06147=1114.760,263.012,-73.129,-178.339,10.074,149.557
C06148=1114.765,262.765,-73.100,-178.342,10.072,149.557
C06149=1114.769,262.516,-73.071,-178.345,10.069,149.557
C06150=1114.773,262.268,-73.041,-178.348,10.066,149.558
C06151=1114.778,262.020,-73.012,-178.351,10.064,149.558
C06152=1114.782,261.771,-72.982,-178.354,10.061,149.558
C06153=1114.786,261.523,-72.954,-178.357,10.058,149.558
C06154=1114.790,261.274,-72.924,-178.360,10.056,149.558
C06155=1114.794,261.027,-72.896,-178.363,10.053,149.558
C06156=1114.799,260.778,-72.867,-178.366,10.050,149.558
C06157=1114.803,260.530,-72.838,-178.369,10.047,149.559
C06158=1114.807,260.282,-72.808,-178.372,10.044,149.559
C06159=1114.812,260.033,-72.779,-178.375,10.041,149.559
C06160=1114.816,259.785,-72.751,-178.378,10.038,149.559
C06161=1114.820,259.537,-72.721,-178.381,10.036,149.559
C06162=1114.824,259.289,-72.692,-178.384,10.032,149.559
C06163=1114.829,259.040,-72.663,-178.387,10.030,149.559
C06164=1114.833,258.792,-72.634,-178.390,10.027,149.559
C06165=1114.837,258.544,-72.606,-178.392,10.024,149.559
C06166=1114.841,258.296,-72.577,-178.395,10.021,149.559
C06167=1114.846,258.047,-72.548,-178.398,10.019,149.559
C06168=1114.849,257.799,-72.519,-178.401,10.016,149.559
C06169=1114.854,257.551,-72.490,-178.404,10.013,149.559
C06170=1114.859,257.302,-72.461,-178.407,10.010,149.560
C06171=1114.863,257.054,-72.432,-178.409,10.008,149.560
C06172=1114.867,256.806,-72.404,-178.412,10.005,149.560
C06173=1114.871,256.558,-72.374,-178.415,10.002,149.560
C06174=1114.876,256.309,-72.346,-178.417,9.999,149.560
C06175=1114.879,256.061,-72.317,-178.420,9.997,149.560
C06176=1114.884,255.812,-72.288,-178.422,9.994,149.560
C06177=1114.889,255.564,-72.260,-178.424,9.993,149.560
C06178=1114.892,255.316,-72.231,-178.425,9.990,149.560
C06179=1114.897,255.067,-72.202,-178.427,9.989,149.560
C06180=1114.902,254.820,-72.173,-178.429,9.987,149.560
C06181=1114.905,254.571,-72.145,-178.431,9.984,149.560
C06182=1114.909,254.323,-72.115,-178.433,9.982,149.560
C06183=1114.913,254.110,-72.092,-178.434,9.981,149.560
C06184=1114.917,253.896,-72.067,-178.436,9.979,149.560
C06185=1114.921,253.684,-72.042,-178.439,9.977,149.560
C06186=1114.924,253.471,-72.018,-178.440,9.975,149.560
C06187=1114.928,253.258,-71.993,-178.442,9.973,149.560
C06188=1114.932,253.045,-71.969,-178.445,9.971,149.560
C06189=1114.935,252.831,-71.944,-178.447,9.969,149.560
C06190=1114.939,252.619,-71.920,-178.449,9.967,149.560
C06191=1114.943,252.370,-71.891,-178.452,9.965,149.561
C06192=1114.948,252.122,-71.863,-178.454,9.963,149.561
C06193=1114.952,251.874,-71.834,-178.457,9.960,149.561
C06194=1114.955,251.625,-71.806,-178.461,9.957,149.561
C06195=1114.961,251.377,-71.777,-178.464,9.955,149.561
C06196=1114.965,251.129,-71.748,-178.467,9.952,149.561
C06197=1114.968,250.880,-71.720,-178.470,9.950,149.562
C06198=1114.974,250.632,-71.691,-178.473,9.947,149.562
C06199=1114.977,250.384,-71.663,-178.477,9.944,149.562
C06200=1114.982,250.135,-71.635,-178.480,9.941,149.562
C06201=1114.986,249.887,-71.607,-178.484,9.938,149.563
C06202=1114.990,249.639,-71.578,-178.488,9.935,149.563
C06203=1114.995,249.391,-71.549,-178.492,9.931,149.563
C06204=1114.998,249.142,-71.521,-178.496,9.928,149.563
C06205=1115.004,248.894,-71.493,-178.499,9.925,149.563
C06206=1115.007,248.645,-71.465,-178.503,9.921,149.564
C06207=1115.012,248.396,-71.436,-178.507,9.918,149.564
C06208=1115.016,248.149,-71.408,-178.512,9.914,149.564
C06209=1115.020,247.900,-71.380,-178.516,9.911,149.564
C06210=1115.025,247.652,-71.352,-178.520,9.906,149.564
C06211=1115.029,247.403,-71.324,-178.523,9.903,149.564
C06212=1115.033,247.155,-71.296,-178.525,9.901,149.564
C06213=1115.038,246.906,-71.267,-178.528,9.898,149.564
C06214=1115.042,246.659,-71.239,-178.530,9.895,149.564
C06215=1115.046,246.410,-71.211,-178.532,9.893,149.564
C06216=1115.051,246.162,-71.183,-178.533,9.891,149.564
C06217=1115.054,245.913,-71.155,-178.536,9.887,149.564
C06218=1115.059,245.665,-71.127,-178.538,9.885,149.564
C06219=1115.063,245.416,-71.098,-178.540,9.883,149.564
C06220=1115.068,245.168,-71.071,-178.543,9.880,149.564
C06221=1115.072,244.919,-71.043,-178.545,9.878,149.564
C06222=1115.077,244.671,-71.014,-178.547,9.875,149.564
C06223=1115.081,244.423,-70.986,-178.549,9.872,149.564
C06224=1115.085,244.175,-70.959,-178.551,9.870,149.564
C06225=1115.089,243.926,-70.930,-178.554,9.867,149.564
C06226=1115.094,243.678,-70.902,-178.556,9.865,149.564
C06227=1115.098,243.429,-70.875,-178.558,9.862,149.564
C06228=1115.102,243.181,-70.847,-178.561,9.860,149.564
C06229=1115.106,242.932,-70.819,-178.563,9.857,149.564
C06230=1115.110,242.684,-70.791,-178.565,9.855,149.564
C06231=1115.116,242.436,-70.763,-178.567,9.852,149.564
C06232=1115.119,242.187,-70.735,-178.570,9.850,149.564
C06233=1115.124,241.939,-70.707,-178.572,9.847,149.564
C06234=1115.127,241.691,-70.679,-178.575,9.844,149.564
C06235=1115.132,241.442,-70.652,-178.577,9.842,149.564
C06236=1115.137,241.193,-70.623,-178.580,9.839,149.564
C06237=1115.141,240.945,-70.596,-178.582,9.837,149.564
C06238=1115.146,240.697,-70.569,-178.585,9.834,149.564
C06239=1115.148,240.484,-70.544,-178.587,9.832,149.564
C06240=1115.152,240.271,-70.520,-178.589,9.830,149.564
C06241=1115.156,240.058,-70.497,-178.591,9.828,149.564
C06242=1115.160,239.844,-70.473,-178.593,9.826,149.564
C06243=1115.164,239.631,-70.449,-178.596,9.824,149.565
C06244=1115.167,239.418,-70.425,-178.597,9.821,149.564
C06245=1115.171,239.205,-70.402,-178.600,9.819,149.565
C06246=1115.174,238.992,-70.378,-178.602,9.817,149.565
C06247=1115.179,238.744,-70.351,-178.605,9.814,149.565
C06248=1115.183,238.495,-70.323,-178.608,9.812,149.565
C06249=1115.188,238.246,-70.295,-178.610,9.810,149.565
C06250=1115.193,237.998,-70.267,-178.613,9.807,149.565
C06251=1115.197,237.749,-70.240,-178.615,9.804,149.565
C06252=1115.201,237.501,-70.212,-178.618,9.802,149.565
C06253=1115.206,237.253,-70.185,-178.621,9.799,149.565
C06254=1115.209,237.004,-70.157,-178.624,9.796,149.565
C06255=1115.214,236.756,-70.130,-178.626,9.794,149.566
C06256=1115.218,236.508,-70.102,-178.628,9.791,149.565
C06257=1115.222,236.259,-70.074,-178.631,9.788,149.566
C06258=1115.227,236.011,-70.047,-178.634,9.786,149.566
C06259=1115.231,235.762,-70.020,-178.637,9.784,149.566
C06260=1115.236,235.513,-69.992,-178.640,9.781,149.566
C06261=1115.240,235.265,-69.964,-178.642,9.778,149.566
C06262=1115.245,235.017,-69.937,-178.645,9.775,149.566
C06263=1115.249,234.769,-69.910,-178.648,9.772,149.566
C06264=1115.253,234.520,-69.882,-178.651,9.770,149.566
C06265=1115.258,234.271,-69.855,-178.654,9.767,149.566
C06266=1115.262,234.023,-69.827,-178.656,9.765,149.567
C06267=1115.266,233.774,-69.800,-178.659,9.762,149.567
C06268=1115.270,233.526,-69.773,-178.662,9.759,149.567
C06269=1115.274,233.278,-69.746,-178.665,9.756,149.567
C06270=1115.279,233.030,-69.719,-178.668,9.754,149.567
C06271=1115.283,232.780,-69.691,-178.670,9.751,149.567
C06272=1115.288,232.532,-69.664,-178.673,9.748,149.567
C06273=1115.292,232.284,-69.636,-178.676,9.745,149.567
C06274=1115.297,232.036,-69.609,-178.679,9.742,149.567
C06275=1115.301,231.787,-69.582,-178.682,9.739,149.567
C06276=1115.305,231.538,-69.555,-178.685,9.736,149.567
C06277=1115.309,231.290,-69.528,-178.688,9.733,149.567
C06278=1115.314,231.042,-69.501,-178.691,9.730,149.568
C06279=1115.318,230.793,-69.473,-178.694,9.727,149.568
C06280=1115.322,230.544,-69.446,-178.697,9.725,149.568
C06281=1115.327,230.296,-69.419,-178.700,9.722,149.568
C06282=1115.331,230.047,-69.393,-178.703,9.718,149.568
C06283=1115.336,229.799,-69.365,-178.706,9.715,149.568
C06284=1115.340,229.550,-69.338,-178.709,9.712,149.568
C06285=1115.345,229.302,-69.311,-178.712,9.710,149.568
C06286=1115.348,229.053,-69.284,-178.715,9.706,149.568
C06287=1115.353,228.805,-69.257,-178.718,9.703,149.568
C06288=1115.358,228.556,-69.230,-178.721,9.700,149.568
C06289=1115.362,228.308,-69.203,-178.723,9.697,149.568
C06290=1115.366,228.059,-69.177,-178.727,9.694,149.568
C06291=1115.371,227.811,-69.150,-178.729,9.691,149.568
C06292=1115.375,227.562,-69.123,-178.732,9.688,149.568
C06293=1115.379,227.314,-69.096,-178.735,9.685,149.568
C06294=1115.383,227.065,-69.069,-178.737,9.682,149.568
C06295=1115.387,226.852,-69.045,-178.740,9.679,149.568
C06296=1115.391,226.638,-69.023,-178.743,9.676,149.568
C06297=1115.394,226.426,-69.000,-178.745,9.673,149.568
C06298=1115.399,226.213,-68.977,-178.748,9.671,149.568
C06299=1115.403,226.000,-68.954,-178.750,9.668,149.568
C06300=1115.407,225.786,-68.931,-178.752,9.665,149.568
C06301=1115.410,225.573,-68.907,-178.754,9.663,149.568
C06302=1115.414,225.360,-68.885,-178.757,9.660,149.568
C06303=1115.418,225.111,-68.858,-178.759,9.657,149.568
C06304=1115.423,224.863,-68.831,-178.762,9.654,149.568
C06305=1115.427,224.615,-68.805,-178.765,9.651,149.568
C06306=1115.431,224.365,-68.778,-178.767,9.648,149.568
C06307=1115.435,224.117,-68.751,-178.770,9.645,149.568
C06308=1115.440,223.868,-68.724,-178.772,9.641,149.568
C06309=1115.444,223.620,-68.698,-178.776,9.638,149.568
C06310=1115.449,223.371,-68.672,-178.778,9.635,149.568
C06311=1115.453,223.123,-68.645,-178.781,9.632,149.568
C06312=1115.457,222.874,-68.618,-178.783,9.629,149.568
C06313=1115.462,222.625,-68.592,-178.786,9.625,149.568
C06314=1115.466,222.377,-68.565,-178.788,9.622,149.568
C06315=1115.471,222.128,-68.538,-178.791,9.619,149.568
C06316=1115.475,221.879,-68.512,-178.793,9.616,149.568
C06317=1115.480,221.631,-68.485,-178.796,9.613,149.567
C06318=1115.484,221.383,-68.459,-178.798,9.610,149.567
C06319=1115.489,221.134,-68.433,-178.801,9.606,149.567
C06320=1115.492,220.885,-68.406,-178.802,9.604,149.567
C06321=1115.496,220.637,-68.380,-178.805,9.601,149.567
C06322=1115.501,220.388,-68.353,-178.807,9.598,149.567
C06323=1115.505,220.140,-68.327,-178.810,9.595,149.567
C06324=1115.511,219.892,-68.301,-178.813,9.592,149.567
C06325=1115.515,219.643,-68.274,-178.815,9.589,149.567
C06326=1115.520,219.394,-68.248,-178.817,9.585,149.567
C06327=1115.524,219.146,-68.222,-178.820,9.582,149.566
C06328=1115.528,218.897,-68.196,-178.822,9.579,149.566
C06329=1115.532,218.649,-68.169,-178.824,9.577,149.566
C06330=1115.537,218.400,-68.143,-178.827,9.573,149.566
C06331=1115.541,218.152,-68.116,-178.829,9.570,149.566
C06332=1115.546,217.903,-68.090,-178.831,9.567,149.566
C06333=1115.549,217.654,-68.064,-178.834,9.564,149.566
C06334=1115.554,217.406,-68.038,-178.836,9.561,149.566
C06335=1115.558,217.157,-68.011,-178.838,9.558,149.566
C06336=1115.563,216.908,-67.985,-178.840,9.555,149.566
C06337=1115.567,216.660,-67.959,-178.842,9.552,149.565
C06338=1115.572,216.412,-67.933,-178.844,9.549,149.565
C06339=1115.576,216.163,-67.907,-178.847,9.546,149.565
C06340=1115.581,215.914,-67.881,-178.849,9.544,149.565
C06341=1115.585,215.666,-67.854,-178.851,9.540,149.565
C06342=1115.589,215.417,-67.828,-178.853,9.537,149.565
C06343=1115.594,215.168,-67.803,-178.855,9.535,149.565
C06344=1115.598,214.920,-67.776,-178.858,9.532,149.565
C06345=1115.603,214.671,-67.750,-178.860,9.528,149.564
C06346=1115.607,214.423,-67.724,-178.862,9.526,149.564
C06347=1115.611,214.174,-67.698,-178.864,9.523,149.564
C06348=1115.615,213.926,-67.672,-178.866,9.520,149.564
C06349=1115.620,213.677,-67.646,-178.868,9.517,149.564
C06350=1115.625,213.428,-67.620,-178.870,9.514,149.564
C06351=1115.629,213.215,-67.598,-178.873,9.511,149.564
C06352=1115.633,213.001,-67.575,-178.875,9.509,149.564
C06353=1115.636,212.788,-67.553,-178.877,9.506,149.564
C06354=1115.640,212.575,-67.530,-178.879,9.504,149.564
C06355=1115.643,212.361,-67.508,-178.881,9.502,149.564
C06356=1115.647,212.149,-67.486,-178.884,9.499,149.564
C06357=1115.652,211.934,-67.464,-178.886,9.496,149.564
C06358=1115.655,211.721,-67.442,-178.888,9.493,149.564
C06359=1115.659,211.472,-67.416,-178.891,9.490,149.564
C06360=1115.664,211.225,-67.390,-178.894,9.487,149.564
C06361=1115.669,210.976,-67.364,-178.896,9.484,149.564
C06362=1115.673,210.727,-67.338,-178.899,9.481,149.564
C06363=1115.677,210.478,-67.313,-178.902,9.478,149.564
C06364=1115.682,210.230,-67.287,-178.904,9.475,149.564
C06365=1115.686,209.981,-67.261,-178.907,9.472,149.564
C06366=1115.690,209.732,-67.236,-178.910,9.469,149.564
C06367=1115.694,209.483,-67.210,-178.913,9.467,149.564
C06368=1115.699,209.235,-67.184,-178.915,9.463,149.564
C06369=1115.704,208.987,-67.159,-178.918,9.461,149.564
C06370=1115.708,208.737,-67.132,-178.921,9.458,149.564
C06371=1115.713,208.489,-67.107,-178.924,9.455,149.564
C06372=1115.718,208.240,-67.081,-178.927,9.452,149.564
C06373=1115.722,207.992,-67.056,-178.929,9.449,149.564
C06374=1115.726,207.743,-67.030,-178.932,9.446,149.564
C06375=1115.731,207.495,-67.004,-178.935,9.444,149.564
C06376=1115.735,207.246,-66.979,-178.938,9.440,149.564
C06377=1115.739,206.997,-66.953,-178.941,9.438,149.565
C06378=1115.744,206.748,-66.928,-178.943,9.435,149.565
C06379=1115.749,206.500,-66.902,-178.946,9.432,149.565
C06380=1115.753,206.251,-66.877,-178.949,9.429,149.565
C06381=1115.758,206.003,-66.851,-178.952,9.426,149.565
C06382=1115.762,205.754,-66.826,-178.955,9.424,149.565
C06383=1115.766,205.505,-66.800,-178.957,9.420,149.565
C06384=1115.771,205.256,-66.775,-178.960,9.418,149.565
C06385=1115.775,205.008,-66.749,-178.963,9.415,149.565
C06386=1115.779,204.759,-66.724,-178.966,9.412,149.565
C06387=1115.784,204.511,-66.699,-178.969,9.409,149.565
C06388=1115.788,204.262,-66.673,-178.972,9.406,149.566
C06389=1115.793,204.013,-66.648,-178.975,9.404,149.566
C06390=1115.797,203.765,-66.623,-178.978,9.401,149.566
C06391=1115.802,203.516,-66.597,-178.980,9.398,149.566
C06392=1115.807,203.267,-66.572,-178.984,9.394,149.566
C06393=1115.811,203.018,-66.547,-178.987,9.392,149.566
C06394=1115.816,202.770,-66.521,-178.990,9.389,149.566
C06395=1115.820,202.521,-66.497,-178.992,9.386,149.566
C06396=1115.824,202.272,-66.471,-178.995,9.383,149.566
C06397=1115.829,202.024,-66.446,-178.998,9.380,149.566
C06398=1115.833,201.775,-66.421,-179.001,9.377,149.566
C06399=1115.838,201.527,-66.395,-179.004,9.374,149.567
C06400=1115.842,201.278,-66.371,-179.007,9.371,149.567
C06401=1115.847,201.029,-66.345,-179.010,9.368,149.567
C06402=1115.851,200.780,-66.320,-179.013,9.365,149.567
C06403=1115.856,200.532,-66.295,-179.015,9.362,149.567
C06404=1115.859,200.283,-66.270,-179.019,9.359,149.567
C06405=1115.864,200.034,-66.245,-179.022,9.356,149.567
C06406=1115.869,199.786,-66.219,-179.025,9.353,149.567
C06407=1115.872,199.572,-66.198,-179.027,9.350,149.567
C06408=1115.877,199.359,-66.177,-179.029,9.348,149.567
C06409=1115.880,199.145,-66.155,-179.032,9.345,149.567
C06410=1115.884,198.931,-66.134,-179.035,9.342,149.567
C06411=1115.888,198.718,-66.112,-179.037,9.339,149.567
C06412=1115.892,198.505,-66.091,-179.040,9.337,149.567
C06413=1115.896,198.291,-66.069,-179.042,9.334,149.567
C06414=1115.900,198.078,-66.048,-179.045,9.331,149.567
C06415=1115.904,197.829,-66.022,-179.048,9.328,149.567
C06416=1115.908,197.580,-65.998,-179.050,9.325,149.567
C06417=1115.913,197.331,-65.973,-179.054,9.321,149.568
C06418=1115.917,197.083,-65.949,-179.056,9.318,149.568
C06419=1115.922,196.835,-65.924,-179.060,9.315,149.568
C06420=1115.927,196.585,-65.899,-179.062,9.312,149.568
C06421=1115.931,196.337,-65.875,-179.065,9.308,149.568
C06422=1115.935,196.088,-65.849,-179.068,9.305,149.568
C06423=1115.940,195.840,-65.825,-179.069,9.303,149.567
C06424=1115.944,195.590,-65.800,-179.071,9.300,149.567
C06425=1115.949,195.342,-65.775,-179.073,9.297,149.567
C06426=1115.953,195.094,-65.750,-179.075,9.294,149.567
C06427=1115.958,194.844,-65.725,-179.077,9.291,149.567
C06428=1115.962,194.596,-65.701,-179.079,9.289,149.567
C06429=1115.967,194.346,-65.676,-179.081,9.286,149.567
C06430=1115.971,194.099,-65.652,-179.083,9.283,149.567
C06431=1115.976,193.850,-65.627,-179.085,9.281,149.566
C06432=1115.980,193.601,-65.602,-179.087,9.278,149.566
C06433=1115.985,193.352,-65.578,-179.089,9.275,149.566
C06434=1115.989,193.103,-65.553,-179.091,9.273,149.566
C06435=1115.994,192.854,-65.529,-179.093,9.269,149.566
C06436=1115.998,192.606,-65.504,-179.095,9.267,149.566
C06437=1116.003,192.357,-65.479,-179.098,9.264,149.566
C06438=1116.007,192.108,-65.455,-179.099,9.262,149.566
C06439=1116.012,191.860,-65.430,-179.101,9.259,149.566
C06440=1116.016,191.611,-65.406,-179.104,9.256,149.566
C06441=1116.021,191.362,-65.381,-179.106,9.254,149.566
C06442=1116.025,191.114,-65.357,-179.108,9.250,149.565
C06443=1116.030,190.864,-65.332,-179.110,9.248,149.565
C06444=1116.034,190.616,-65.308,-179.112,9.245,149.565
C06445=1116.039,190.367,-65.283,-179.114,9.242,149.565
C06446=1116.043,190.118,-65.259,-179.117,9.239,149.565
C06447=1116.048,189.869,-65.234,-179.119,9.236,149.565
C06448=1116.053,189.621,-65.210,-179.121,9.234,149.565
C06449=1116.057,189.372,-65.185,-179.124,9.231,149.565
C06450=1116.062,189.123,-65.161,-179.126,9.228,149.565
C06451=1116.066,188.874,-65.137,-179.128,9.225,149.565
C06452=1116.071,188.625,-65.112,-179.130,9.223,149.565
C06453=1116.075,188.377,-65.088,-179.132,9.220,149.565
C06454=1116.079,188.128,-65.064,-179.135,9.217,149.565
C06455=1116.085,187.879,-65.039,-179.137,9.215,149.565
C06456=1116.088,187.630,-65.014,-179.139,9.211,149.565
C06457=1116.093,187.382,-64.990,-179.142,9.208,149.565
C06458=1116.098,187.133,-64.966,-179.144,9.206,149.565
C06459=1116.103,186.884,-64.942,-179.146,9.203,149.565
C06460=1116.106,186.635,-64.918,-179.149,9.200,149.565
C06461=1116.111,186.386,-64.893,-179.151,9.197,149.565
C06462=1116.116,186.138,-64.869,-179.153,9.194,149.565
C06463=1116.120,185.924,-64.849,-179.156,9.192,149.565
C06464=1116.123,185.710,-64.828,-179.158,9.189,149.565
C06465=1116.127,185.497,-64.807,-179.160,9.187,149.565
C06466=1116.132,185.283,-64.786,-179.162,9.185,149.565
C06467=1116.135,185.070,-64.765,-179.164,9.182,149.565
C06468=1116.139,184.856,-64.745,-179.166,9.180,149.565
C06469=1116.143,184.643,-64.725,-179.168,9.177,149.565
C06470=1116.146,184.429,-64.703,-179.170,9.174,149.564
C06471=1116.151,184.180,-64.680,-179.173,9.171,149.564
C06472=1116.156,183.931,-64.655,-179.175,9.168,149.564
C06473=1116.161,183.683,-64.631,-179.178,9.165,149.564
C06474=1116.165,183.434,-64.608,-179.180,9.163,149.564
C06475=1116.170,183.185,-64.584,-179.182,9.160,149.564
C06476=1116.174,182.936,-64.559,-179.185,9.157,149.564
C06477=1116.179,182.687,-64.535,-179.188,9.154,149.564
C06478=1116.183,182.438,-64.511,-179.190,9.151,149.564
C06479=1116.188,182.190,-64.487,-179.193,9.148,149.564
C06480=1116.192,181.941,-64.464,-179.195,9.145,149.564
C06481=1116.197,181.693,-64.440,-179.198,9.141,149.564
C06482=1116.201,181.443,-64.415,-179.200,9.138,149.564
C06483=1116.205,181.194,-64.392,-179.203,9.135,149.564
C06484=1116.211,180.946,-64.367,-179.205,9.132,149.564
C06485=1116.215,180.697,-64.344,-179.208,9.129,149.564
C06486=1116.220,180.448,-64.320,-179.210,9.126,149.564
C06487=1116.224,180.199,-64.296,-179.213,9.123,149.564
C06488=1116.229,179.951,-64.272,-179.215,9.120,149.564
C06489=1116.233,179.701,-64.249,-179.218,9.117,149.564
C06490=1116.237,179.453,-64.224,-179.220,9.113,149.564
C06491=1116.242,179.204,-64.201,-179.223,9.110,149.564
C06492=1116.246,178.955,-64.177,-179.225,9.107,149.564
C06493=1116.251,178.706,-64.154,-179.228,9.104,149.563
C06494=1116.255,178.458,-64.130,-179.229,9.101,149.563
C06495=1116.260,178.209,-64.106,-179.232,9.098,149.563
C06496=1116.265,177.960,-64.083,-179.234,9.095,149.563
C06497=1116.269,177.711,-64.059,-179.236,9.092,149.563
C06498=1116.274,177.462,-64.035,-179.238,9.089,149.563
C06499=1116.278,177.214,-64.011,-179.240,9.087,149.563
C06500=1116.283,176.965,-63.988,-179.242,9.084,149.563
C06501=1116.288,176.716,-63.965,-179.245,9.080,149.563
C06502=1116.292,176.467,-63.941,-179.246,9.078,149.563
C06503=1116.297,176.218,-63.917,-179.249,9.075,149.562
C06504=1116.301,175.969,-63.893,-179.251,9.072,149.562
C06505=1116.305,175.720,-63.869,-179.253,9.069,149.562
C06506=1116.310,175.471,-63.846,-179.255,9.066,149.562
C06507=1116.315,175.222,-63.823,-179.258,9.063,149.562
C06508=1116.319,174.973,-63.799,-179.259,9.060,149.562
C06509=1116.324,174.725,-63.775,-179.262,9.057,149.562
C06510=1116.328,174.476,-63.752,-179.264,9.054,149.562
C06511=1116.333,174.227,-63.729,-179.266,9.051,149.562
C06512=1116.337,173.978,-63.706,-179.268,9.048,149.562
C06513=1116.341,173.729,-63.682,-179.271,9.045,149.561
C06514=1116.346,173.480,-63.658,-179.272,9.042,149.561
C06515=1116.351,173.231,-63.635,-179.275,9.039,149.561
C06516=1116.356,172.983,-63.612,-179.277,9.036,149.561
C06517=1116.361,172.734,-63.589,-179.280,9.033,149.561
C06518=1116.366,172.485,-63.565,-179.281,9.030,149.561
C06519=1116.368,172.271,-63.544,-179.283,9.028,149.561
C06520=1116.372,172.058,-63.525,-179.286,9.025,149.561
C06521=1116.377,171.844,-63.504,-179.287,9.022,149.561
C06522=1116.381,171.630,-63.484,-179.289,9.020,149.561
C06523=1116.384,171.417,-63.465,-179.291,9.017,149.561
C06524=1116.388,171.203,-63.445,-179.293,9.015,149.561
C06525=1116.393,170.989,-63.424,-179.295,9.011,149.560
C06526=1116.396,170.776,-63.405,-179.297,9.009,149.560
C06527=1116.401,170.527,-63.381,-179.299,9.007,149.560
C06528=1116.406,170.278,-63.358,-179.301,9.004,149.560
C06529=1116.410,170.029,-63.335,-179.304,9.000,149.560
C06530=1116.414,169.780,-63.312,-179.306,8.997,149.560
C06531=1116.419,169.531,-63.288,-179.308,8.995,149.560
C06532=1116.424,169.282,-63.265,-179.310,8.991,149.560
C06533=1116.428,169.034,-63.243,-179.313,8.988,149.560
C06534=1116.433,168.785,-63.219,-179.315,8.985,149.560
C06535=1116.438,168.536,-63.196,-179.317,8.982,149.559
C06536=1116.443,168.287,-63.173,-179.319,8.979,149.559
C06537=1116.446,168.038,-63.150,-179.322,8.976,149.559
C06538=1116.451,167.788,-63.127,-179.324,8.973,149.559
C06539=1116.456,167.539,-63.104,-179.326,8.970,149.559
C06540=1116.461,167.291,-63.081,-179.328,8.967,149.559
C06541=1116.465,167.042,-63.058,-179.330,8.964,149.559
C06542=1116.470,166.793,-63.035,-179.333,8.961,149.559
C06543=1116.474,166.545,-63.012,-179.335,8.957,149.559
C06544=1116.479,166.296,-62.989,-179.337,8.955,149.558
C06545=1116.483,166.047,-62.965,-179.339,8.952,149.558
C06546=1116.488,165.798,-62.944,-179.342,8.949,149.558
C06547=1116.493,165.549,-62.920,-179.344,8.945,149.558
C06548=1116.498,165.300,-62.897,-179.346,8.942,149.558
C06549=1116.502,165.051,-62.874,-179.348,8.939,149.558
C06550=1116.506,164.802,-62.851,-179.350,8.936,149.558
C06551=1116.511,164.553,-62.829,-179.353,8.933,149.558
C06552=1116.516,164.304,-62.806,-179.355,8.930,149.557
C06553=1116.521,164.055,-62.782,-179.357,8.926,149.557
C06554=1116.525,163.807,-62.759,-179.359,8.923,149.557
C06555=1116.530,163.557,-62.737,-179.362,8.920,149.557
C06556=1116.534,163.309,-62.714,-179.364,8.917,149.557
C06557=1116.539,163.060,-62.691,-179.366,8.914,149.557
C06558=1116.543,162.811,-62.669,-179.369,8.911,149.557
C06559=1116.548,162.562,-62.646,-179.371,8.907,149.557
C06560=1116.552,162.313,-62.623,-179.373,8.904,149.557
C06561=1116.557,162.064,-62.601,-179.376,8.901,149.557
C06562=1116.561,161.815,-62.578,-179.378,8.898,149.556
C06563=1116.566,161.566,-62.555,-179.380,8.895,149.556
C06564=1116.571,161.318,-62.533,-179.382,8.892,149.556
C06565=1116.576,161.068,-62.509,-179.384,8.889,149.556
C06566=1116.580,160.820,-62.487,-179.386,8.885,149.556
C06567=1116.585,160.570,-62.464,-179.389,8.882,149.556
C06568=1116.589,160.322,-62.442,-179.391,8.879,149.556
C06569=1116.594,160.072,-62.419,-179.393,8.876,149.555
C06570=1116.598,159.824,-62.396,-179.396,8.872,149.555
C06571=1116.604,159.575,-62.374,-179.398,8.869,149.555
C06572=1116.608,159.326,-62.351,-179.401,8.866,149.555
C06573=1116.612,159.077,-62.329,-179.403,8.862,149.555
C06574=1116.617,158.828,-62.306,-179.405,8.859,149.555
C06575=1116.621,158.614,-62.287,-179.407,8.857,149.555
C06576=1116.625,158.401,-62.267,-179.409,8.854,149.555
C06577=1116.629,158.186,-62.248,-179.411,8.851,149.554
C06578=1116.633,157.973,-62.228,-179.412,8.848,149.554
C06579=1116.636,157.759,-62.210,-179.415,8.845,149.554
C06580=1116.640,157.545,-62.191,-179.416,8.843,149.554
C06581=1116.644,157.331,-62.171,-179.419,8.839,149.554
C06582=1116.648,157.117,-62.152,-179.420,8.837,149.554
C06583=1116.653,156.868,-62.130,-179.423,8.833,149.554
C06584=1116.658,156.619,-62.107,-179.425,8.830,149.554
C06585=1116.663,156.371,-62.085,-179.427,8.827,149.553
C06586=1116.667,156.122,-62.062,-179.429,8.823,149.553
C06587=1116.672,155.872,-62.040,-179.432,8.820,149.553
C06588=1116.677,155.624,-62.018,-179.434,8.817,149.553
C06589=1116.681,155.375,-61.995,-179.436,8.814,149.553
C06590=1116.686,155.126,-61.973,-179.438,8.810,149.553
C06591=1116.690,154.877,-61.951,-179.440,8.807,149.552
C06592=1116.695,154.627,-61.929,-179.443,8.803,149.552
C06593=1116.699,154.379,-61.907,-179.445,8.800,149.552
C06594=1116.704,154.130,-61.884,-179.447,8.796,149.552
C06595=1116.709,153.881,-61.862,-179.450,8.793,149.552
C06596=1116.713,153.632,-61.840,-179.452,8.790,149.552
C06597=1116.717,153.383,-61.817,-179.454,8.786,149.551
C06598=1116.723,153.134,-61.795,-179.457,8.782,149.551
C06599=1116.727,152.885,-61.773,-179.459,8.779,149.551
C06600=1116.732,152.636,-61.751,-179.461,8.775,149.551
C06601=1116.736,152.387,-61.729,-179.463,8.772,149.551
C06602=1116.741,152.138,-61.708,-179.466,8.769,149.551
C06603=1116.746,151.889,-61.684,-179.468,8.765,149.550
C06604=1116.751,151.640,-61.663,-179.470,8.762,149.550
C06605=1116.755,151.391,-61.641,-179.472,8.758,149.550
C06606=1116.760,151.142,-61.619,-179.475,8.755,149.550
C06607=1116.764,150.893,-61.597,-179.477,8.751,149.550
C06608=1116.769,150.644,-61.575,-179.479,8.748,149.549
C06609=1116.774,150.395,-61.553,-179.481,8.744,149.549
C06610=1116.779,150.146,-61.531,-179.484,8.741,149.549
C06611=1116.783,149.897,-61.509,-179.486,8.737,149.549
C06612=1116.788,149.648,-61.487,-179.489,8.733,149.549
C06613=1116.792,149.399,-61.465,-179.491,8.730,149.548
C06614=1116.797,149.150,-61.443,-179.493,8.726,149.548
C06615=1116.802,148.901,-61.421,-179.495,8.723,149.548
C06616=1116.806,148.652,-61.400,-179.498,8.718,149.548
C06617=1116.811,148.404,-61.378,-179.500,8.715,149.547
C06618=1116.816,148.154,-61.356,-179.502,8.712,149.547
C06619=1116.820,147.906,-61.334,-179.504,8.708,149.547
C06620=1116.825,147.656,-61.312,-179.506,8.705,149.547
C06621=1116.830,147.408,-61.291,-179.509,8.700,149.546
C06622=1116.834,147.158,-61.269,-179.511,8.697,149.546
C06623=1116.839,146.910,-61.247,-179.513,8.693,149.546
C06624=1116.844,146.660,-61.226,-179.516,8.689,149.546
C06625=1116.848,146.411,-61.204,-179.518,8.686,149.546
C06626=1116.853,146.162,-61.182,-179.520,8.682,149.545
C06627=1116.857,145.913,-61.160,-179.522,8.679,149.545
C06628=1116.862,145.664,-61.138,-179.525,8.674,149.545
C06629=1116.867,145.415,-61.117,-179.527,8.671,149.545
C06630=1116.872,145.166,-61.095,-179.529,8.667,149.544
C06631=1116.876,144.952,-61.077,-179.530,8.663,149.544
C06632=1116.880,144.738,-61.058,-179.532,8.661,149.544
C06633=1116.884,144.524,-61.039,-179.533,8.658,149.543
C06634=1116.888,144.311,-61.022,-179.534,8.655,149.543
C06635=1116.892,144.096,-61.003,-179.536,8.652,149.543
C06636=1116.896,143.882,-60.983,-179.537,8.650,149.543
C06637=1116.900,143.669,-60.965,-179.538,8.646,149.542
C06638=1116.904,143.455,-60.946,-179.540,8.644,149.542
C06639=1116.909,143.206,-60.926,-179.542,8.640,149.542
C06640=1116.913,142.956,-60.904,-179.543,8.637,149.541
C06641=1116.918,142.708,-60.882,-179.545,8.634,149.541
C06642=1116.923,142.459,-60.861,-179.546,8.630,149.541
C06643=1116.927,142.209,-60.839,-179.548,8.627,149.540
C06644=1116.932,141.961,-60.817,-179.549,8.623,149.540
C06645=1116.936,141.712,-60.797,-179.552,8.620,149.540
C06646=1116.941,141.462,-60.775,-179.553,8.617,149.539
C06647=1116.946,141.213,-60.754,-179.555,8.613,149.539
C06648=1116.951,140.964,-60.732,-179.556,8.610,149.539
C06649=1116.956,140.716,-60.711,-179.558,8.607,149.538
C06650=1116.960,140.466,-60.689,-179.559,8.603,149.538
C06651=1116.964,140.217,-60.668,-179.561,8.600,149.538
C06652=1116.970,139.968,-60.647,-179.562,8.596,149.537
C06653=1116.974,139.719,-60.625,-179.564,8.593,149.537
C06654=1116.979,139.470,-60.604,-179.566,8.590,149.537
C06655=1116.983,139.221,-60.583,-179.568,8.586,149.536
C06656=1116.988,138.973,-60.562,-179.569,8.583,149.536
C06657=1116.993,138.723,-60.540,-179.571,8.579,149.536
C06658=1116.997,138.474,-60.519,-179.573,8.576,149.535
C06659=1117.002,138.225,-60.498,-179.574,8.573,149.535
C06660=1117.007,137.976,-60.477,-179.576,8.569,149.535
C06661=1117.011,137.727,-60.455,-179.577,8.567,149.535
C06662=1117.016,137.477,-60.434,-179.579,8.563,149.534
C06663=1117.021,137.229,-60.413,-179.581,8.559,149.534
C06664=1117.026,136.980,-60.392,-179.582,8.557,149.534
C06665=1117.030,136.730,-60.370,-179.584,8.553,149.533
C06666=1117.034,136.481,-60.350,-179.586,8.549,149.533
C06667=1117.039,136.233,-60.328,-179.588,8.547,149.533
C06668=1117.045,135.983,-60.307,-179.589,8.543,149.532
C06669=1117.049,135.735,-60.287,-179.591,8.540,149.532
C06670=1117.053,135.485,-60.265,-179.592,8.536,149.532
C06671=1117.058,135.236,-60.244,-179.594,8.533,149.531
C06672=1117.063,134.987,-60.223,-179.596,8.530,149.531
C06673=1117.068,134.738,-60.202,-179.597,8.526,149.531
C06674=1117.073,134.489,-60.181,-179.600,8.522,149.531
C06675=1117.077,134.240,-60.160,-179.601,8.520,149.530
C06676=1117.082,133.991,-60.138,-179.603,8.516,149.530
C06677=1117.086,133.742,-60.118,-179.605,8.512,149.530
C06678=1117.091,133.493,-60.097,-179.606,8.510,149.529
C06679=1117.096,133.243,-60.076,-179.608,8.506,149.529
C06680=1117.100,132.995,-60.055,-179.609,8.503,149.529
C06681=1117.106,132.746,-60.034,-179.611,8.500,149.529
C06682=1117.109,132.496,-60.013,-179.613,8.496,149.528
C06683=1117.115,132.247,-59.992,-179.614,8.493,149.528
C06684=1117.120,131.998,-59.970,-179.616,8.490,149.528
C06685=1117.124,131.749,-59.950,-179.618,8.486,149.527
C06686=1117.129,131.500,-59.929,-179.620,8.483,149.527
C06687=1117.133,131.285,-59.911,-179.621,8.480,149.527
C06688=1117.137,131.072,-59.893,-179.623,8.477,149.527
C06689=1117.141,130.859,-59.876,-179.624,8.474,149.526
C06690=1117.145,130.644,-59.857,-179.626,8.471,149.526
C06691=1117.150,130.430,-59.840,-179.627,8.469,149.526
C06692=1117.153,130.216,-59.822,-179.629,8.466,149.526
C06693=1117.157,130.002,-59.804,-179.630,8.463,149.525
C06694=1117.161,129.788,-59.786,-179.632,8.460,149.525
C06695=1117.166,129.539,-59.765,-179.633,8.457,149.525
C06696=1117.171,129.290,-59.745,-179.635,8.453,149.525
C06697=1117.176,129.040,-59.724,-179.637,8.450,149.524
C06698=1117.180,128.791,-59.704,-179.639,8.447,149.524
C06699=1117.185,128.542,-59.683,-179.641,8.443,149.524
C06700=1117.189,128.294,-59.662,-179.642,8.440,149.523
C06701=1117.195,128.045,-59.641,-179.644,8.437,149.523
C06702=1117.199,127.796,-59.620,-179.646,8.433,149.523
C06703=1117.203,127.547,-59.600,-179.647,8.430,149.523
C06704=1117.209,127.297,-59.579,-179.649,8.427,149.522
C06705=1117.213,127.048,-59.559,-179.651,8.423,149.522
C06706=1117.218,126.799,-59.538,-179.653,8.420,149.522
C06707=1117.223,126.550,-59.517,-179.654,8.417,149.521
C06708=1117.227,126.301,-59.497,-179.656,8.413,149.521
C06709=1117.233,126.051,-59.477,-179.658,8.410,149.521
C06710=1117.237,125.802,-59.456,-179.660,8.407,149.521
C06711=1117.242,125.553,-59.435,-179.662,8.403,149.520
C06712=1117.247,125.304,-59.415,-179.664,8.400,149.520
C06713=1117.251,125.055,-59.395,-179.665,8.397,149.520
C06714=1117.256,124.806,-59.374,-179.667,8.393,149.520
C06715=1117.261,124.557,-59.353,-179.669,8.390,149.519
C06716=1117.265,124.308,-59.333,-179.670,8.387,149.519
C06717=1117.270,124.059,-59.312,-179.672,8.383,149.519
C06718=1117.275,123.810,-59.292,-179.674,8.380,149.518
C06719=1117.280,123.560,-59.272,-179.676,8.377,149.518
C06720=1117.284,123.311,-59.251,-179.677,8.373,149.518
C06721=1117.289,123.062,-59.231,-179.679,8.370,149.518
C06722=1117.294,122.813,-59.210,-179.681,8.366,149.517
C06723=1117.298,122.564,-59.190,-179.683,8.363,149.517
C06724=1117.303,122.314,-59.170,-179.685,8.360,149.517
C06725=1117.308,122.065,-59.149,-179.687,8.356,149.516
C06726=1117.312,121.816,-59.129,-179.688,8.353,149.516
C06727=1117.317,121.567,-59.108,-179.690,8.350,149.516
C06728=1117.322,121.318,-59.087,-179.692,8.346,149.516
C06729=1117.327,121.069,-59.068,-179.694,8.342,149.515
C06730=1117.331,120.820,-59.047,-179.695,8.340,149.515
C06731=1117.336,120.571,-59.027,-179.697,8.336,149.515
C06732=1117.340,120.321,-59.007,-179.699,8.333,149.515
C06733=1117.346,120.073,-58.987,-179.701,8.329,149.514
C06734=1117.351,119.824,-58.966,-179.702,8.326,149.514
C06735=1117.355,119.574,-58.947,-179.704,8.323,149.514
C06736=1117.360,119.325,-58.926,-179.707,8.319,149.514
C06737=1117.364,119.076,-58.906,-179.708,8.316,149.513
C06738=1117.369,118.827,-58.886,-179.710,8.313,149.513
C06739=1117.374,118.577,-58.865,-179.712,8.309,149.513
C06740=1117.378,118.328,-58.845,-179.714,8.306,149.512
C06741=1117.383,118.079,-58.825,-179.716,8.302,149.512
C06742=1117.388,117.831,-58.805,-179.717,8.299,149.512
C06743=1117.395,117.479,-58.776,-179.720,8.294,149.512
C06744=1117.401,117.128,-58.749,-179.722,8.289,149.511
C06745=1117.408,116.777,-58.721,-179.725,8.285,149.511
C06746=1117.415,116.425,-58.692,-179.727,8.279,149.510
C06747=1117.420,116.176,-58.673,-179.729,8.276,149.510
C06748=1117.425,115.927,-58.652,-179.731,8.273,149.510
C06749=1117.429,115.678,-58.633,-179.733,8.269,149.509
C06750=1117.434,115.429,-58.612,-179.735,8.266,149.509
C06751=1117.439,115.179,-58.593,-179.737,8.262,149.509
C06752=1117.444,114.931,-58.573,-179.738,8.259,149.509
C06753=1117.448,114.681,-58.553,-179.740,8.255,149.508
C06754=1117.453,114.432,-58.533,-179.742,8.252,149.508
C06755=1117.458,114.183,-58.513,-179.744,8.248,149.508
C06756=1117.462,113.934,-58.492,-179.746,8.245,149.508
C06757=1117.467,113.685,-58.473,-179.747,8.242,149.507
C06758=1117.472,113.435,-58.454,-179.749,8.238,149.507
C06759=1117.477,113.187,-58.433,-179.751,8.235,149.507
C06760=1117.481,112.937,-58.414,-179.753,8.231,149.506
C06761=1117.487,112.688,-58.394,-179.755,8.227,149.506
C06762=1117.491,112.439,-58.374,-179.756,8.225,149.506
C06763=1117.496,112.190,-58.354,-179.758,8.221,149.506
C06764=1117.501,111.940,-58.335,-179.760,8.217,149.505
C06765=1117.506,111.692,-58.315,-179.762,8.214,149.505
C06766=1117.510,111.442,-58.295,-179.764,8.210,149.505
C06767=1117.515,111.193,-58.275,-179.766,8.207,149.504
C06768=1117.520,110.944,-58.255,-179.768,8.203,149.504
C06769=1117.525,110.695,-58.236,-179.770,8.200,149.504
C06770=1117.530,110.445,-58.216,-179.772,8.196,149.504
C06771=1117.534,110.196,-58.196,-179.774,8.193,149.503
C06772=1117.539,109.947,-58.178,-179.776,8.188,149.503
C06773=1117.543,109.698,-58.157,-179.779,8.185,149.503
C06774=1117.548,109.449,-58.138,-179.781,8.181,149.503
C06775=1117.554,109.200,-58.118,-179.783,8.177,149.502
C06776=1117.558,108.950,-58.099,-179.785,8.173,149.502
C06777=1117.563,108.701,-58.079,-179.787,8.170,149.502
C06778=1117.568,108.452,-58.059,-179.789,8.166,149.502
C06779=1117.572,108.203,-58.040,-179.792,8.162,149.501
C06780=1117.577,107.954,-58.020,-179.793,8.158,149.501
C06781=1117.582,107.705,-58.001,-179.795,8.154,149.501
C06782=1117.587,107.455,-57.981,-179.797,8.151,149.501
C06783=1117.592,107.206,-57.962,-179.800,8.147,149.500
C06784=1117.596,106.957,-57.943,-179.802,8.143,149.500
C06785=1117.601,106.707,-57.923,-179.804,8.139,149.500
C06786=1117.606,106.459,-57.904,-179.806,8.136,149.499
C06787=1117.612,106.132,-57.878,-179.809,8.130,149.499
C06788=1117.618,105.806,-57.853,-179.811,8.126,149.499
C06789=1117.624,105.480,-57.827,-179.814,8.120,149.498
C06790=1117.631,105.154,-57.802,-179.816,8.115,149.498
C06791=1117.636,104.904,-57.783,-179.818,8.112,149.497
C06792=1117.640,104.655,-57.764,-179.820,8.107,149.497
C06793=1117.646,104.406,-57.744,-179.822,8.104,149.497
C06794=1117.650,104.156,-57.725,-179.824,8.100,149.497
C06795=1117.654,103.942,-57.709,-179.825,8.097,149.496
C06796=1117.659,103.728,-57.692,-179.827,8.094,149.496
C06797=1117.662,103.514,-57.676,-179.829,8.090,149.496
C06798=1117.667,103.299,-57.659,-179.830,8.087,149.495
C06799=1117.671,103.086,-57.642,-179.833,8.084,149.495
C06800=1117.675,102.871,-57.626,-179.834,8.081,149.495
C06801=1117.679,102.657,-57.610,-179.836,8.077,149.494
C06802=1117.684,102.443,-57.593,-179.837,8.074,149.494
C06803=1117.688,102.194,-57.574,-179.839,8.070,149.494
C06804=1117.693,101.944,-57.555,-179.841,8.066,149.494
C06805=1117.698,101.695,-57.536,-179.843,8.062,149.493
C06806=1117.703,101.446,-57.517,-179.844,8.058,149.493
C06807=1117.707,101.196,-57.497,-179.847,8.055,149.492
C06808=1117.712,100.948,-57.479,-179.848,8.051,149.492
C06809=1117.717,100.698,-57.460,-179.850,8.047,149.492
C06810=1117.722,100.449,-57.441,-179.852,8.044,149.491
C06811=1117.726,100.200,-57.421,-179.853,8.040,149.491
C06812=1117.732,99.951,-57.402,-179.856,8.035,149.490
C06813=1117.736,99.701,-57.384,-179.857,8.031,149.490
C06814=1117.741,99.452,-57.364,-179.859,8.028,149.490
C06815=1117.745,99.203,-57.345,-179.861,8.024,149.489
C06816=1117.751,98.953,-57.327,-179.862,8.020,149.489
C06817=1117.756,98.705,-57.308,-179.864,8.016,149.489
C06818=1117.760,98.455,-57.288,-179.866,8.012,149.488
C06819=1117.765,98.206,-57.270,-179.868,8.009,149.488
C06820=1117.770,97.956,-57.251,-179.869,8.005,149.487
C06821=1117.775,97.708,-57.232,-179.871,8.001,149.487
C06822=1117.780,97.458,-57.213,-179.873,7.997,149.487
C06823=1117.784,97.209,-57.194,-179.874,7.993,149.486
C06824=1117.789,96.960,-57.176,-179.876,7.989,149.486
C06825=1117.794,96.710,-57.157,-179.877,7.985,149.485
C06826=1117.799,96.461,-57.139,-179.879,7.981,149.485
C06827=1117.803,96.212,-57.119,-179.881,7.978,149.485
C06828=1117.808,95.963,-57.100,-179.883,7.974,149.484
C06829=1117.814,95.713,-57.082,-179.884,7.970,149.484
C06830=1117.818,95.464,-57.063,-179.886,7.966,149.483
C06831=1117.823,95.215,-57.045,-179.887,7.962,149.483
C06832=1117.827,94.965,-57.025,-179.889,7.958,149.482
C06833=1117.832,94.716,-57.007,-179.891,7.954,149.482
C06834=1117.838,94.467,-56.989,-179.892,7.951,149.482
C06835=1117.842,94.218,-56.970,-179.894,7.947,149.481
C06836=1117.847,93.968,-56.952,-179.895,7.943,149.481
C06837=1117.852,93.720,-56.932,-179.897,7.939,149.480
C06838=1117.857,93.470,-56.914,-179.898,7.935,149.480
C06839=1117.861,93.221,-56.895,-179.900,7.931,149.479
C06840=1117.867,92.972,-56.877,-179.901,7.928,149.479
C06841=1117.871,92.722,-56.858,-179.902,7.924,149.478
C06842=1117.876,92.473,-56.840,-179.904,7.920,149.478
C06843=1117.881,92.224,-56.821,-179.906,7.916,149.478
C06844=1117.885,91.974,-56.802,-179.907,7.912,149.477
C06845=1117.890,91.725,-56.784,-179.909,7.908,149.477
C06846=1117.896,91.476,-56.765,-179.910,7.904,149.476
C06847=1117.901,91.227,-56.747,-179.911,7.900,149.476
C06848=1117.905,90.977,-56.728,-179.913,7.896,149.475
C06849=1117.910,90.728,-56.710,-179.914,7.893,149.475
C06850=1117.915,90.479,-56.692,-179.916,7.889,149.474
C06851=1117.919,90.265,-56.676,-179.917,7.885,149.474
C06852=1117.923,90.050,-56.660,-179.918,7.882,149.473
C06853=1117.927,89.836,-56.644,-179.919,7.879,149.473
C06854=1117.931,89.622,-56.628,-179.920,7.876,149.473
C06855=1117.935,89.407,-56.613,-179.922,7.872,149.472
C06856=1117.940,89.193,-56.596,-179.923,7.869,149.472
C06857=1117.944,88.978,-56.581,-179.924,7.866,149.471
C06858=1117.948,88.764,-56.565,-179.926,7.862,149.471
C06859=1117.953,88.515,-56.547,-179.926,7.859,149.470
C06860=1117.957,88.265,-56.529,-179.928,7.855,149.470
C06861=1117.962,88.016,-56.511,-179.929,7.851,149.470
C06862=1117.968,87.767,-56.491,-179.931,7.847,149.469
C06863=1117.973,87.518,-56.473,-179.931,7.844,149.468
C06864=1117.977,87.268,-56.455,-179.933,7.840,149.468
C06865=1117.982,87.019,-56.437,-179.935,7.836,149.468
C06866=1117.987,86.770,-56.419,-179.936,7.832,149.467
C06867=1117.992,86.521,-56.401,-179.937,7.828,149.467
C06868=1117.997,86.272,-56.383,-179.938,7.825,149.466
C06869=1118.001,86.022,-56.363,-179.940,7.820,149.465
C06870=1118.006,85.773,-56.345,-179.941,7.816,149.465
C06871=1118.011,85.524,-56.327,-179.942,7.813,149.464
C06872=1118.016,85.274,-56.310,-179.943,7.809,149.464
C06873=1118.021,85.025,-56.292,-179.945,7.805,149.464
C06874=1118.026,84.776,-56.274,-179.945,7.802,149.463
C06875=1118.030,84.526,-56.255,-179.947,7.798,149.462
C06876=1118.035,84.277,-56.237,-179.948,7.793,149.462
C06877=1118.040,84.028,-56.219,-179.949,7.790,149.461
C06878=1118.045,83.779,-56.201,-179.951,7.786,149.461
C06879=1118.050,83.529,-56.183,-179.952,7.782,149.460
C06880=1118.055,83.280,-56.165,-179.953,7.779,149.460
C06881=1118.060,83.030,-56.146,-179.954,7.775,149.459
C06882=1118.065,82.781,-56.128,-179.955,7.771,149.459
C06883=1118.070,82.532,-56.110,-179.956,7.767,149.458
C06884=1118.075,82.283,-56.092,-179.957,7.763,149.458
C06885=1118.079,82.033,-56.074,-179.958,7.760,149.457
C06886=1118.084,81.784,-56.056,-179.960,7.756,149.457
C06887=1118.089,81.535,-56.038,-179.961,7.752,149.456
C06888=1118.094,81.286,-56.021,-179.962,7.749,149.456
C06889=1118.098,81.036,-56.002,-179.963,7.745,149.455
C06890=1118.104,80.786,-55.985,-179.964,7.741,149.454
C06891=1118.109,80.537,-55.967,-179.965,7.737,149.454
C06892=1118.114,80.288,-55.949,-179.966,7.734,149.453
C06893=1118.118,80.039,-55.931,-179.967,7.730,149.453
C06894=1118.123,79.790,-55.913,-179.968,7.726,149.452
C06895=1118.128,79.541,-55.896,-179.969,7.722,149.452
C06896=1118.132,79.291,-55.878,-179.970,7.719,149.451
C06897=1118.138,79.042,-55.860,-179.971,7.715,149.451
C06898=1118.143,78.793,-55.842,-179.972,7.712,149.450
C06899=1118.147,78.543,-55.824,-179.973,7.707,149.450
C06900=1118.152,78.294,-55.806,-179.974,7.704,149.449
C06901=1118.157,78.044,-55.788,-179.975,7.700,149.448
C06902=1118.162,77.794,-55.771,-179.976,7.697,149.448
C06903=1118.167,77.545,-55.753,-179.977,7.693,149.447
C06904=1118.172,77.296,-55.735,-179.978,7.689,149.447
C06905=1118.177,77.047,-55.717,-179.980,7.685,149.446
C06906=1118.182,76.797,-55.700,-179.980,7.682,149.446
C06907=1118.186,76.584,-55.684,-179.982,7.678,149.445
C06908=1118.190,76.369,-55.669,-179.983,7.675,149.445
C06909=1118.194,76.155,-55.654,-179.984,7.672,149.444
C06910=1118.199,75.941,-55.639,-179.985,7.668,149.444
C06911=1118.203,75.726,-55.623,-179.986,7.665,149.444
C06912=1118.207,75.511,-55.608,-179.987,7.662,149.443
C06913=1118.212,75.297,-55.593,-179.989,7.658,149.443
C06914=1118.215,75.083,-55.578,-179.990,7.655,149.442
C06915=1118.220,74.834,-55.560,-179.991,7.651,149.442
C06916=1118.225,74.584,-55.543,-179.993,7.647,149.441
C06917=1118.230,74.335,-55.525,-179.994,7.643,149.441
C06918=1118.235,74.085,-55.508,-179.996,7.639,149.440
C06919=1118.239,73.836,-55.490,-179.997,7.635,149.440
C06920=1118.244,73.587,-55.472,-179.999,7.631,149.439
C06921=1118.249,73.337,-55.455,180.000,7.627,149.439
C06922=1118.254,73.088,-55.437,179.998,7.623,149.439
C06923=1118.259,72.838,-55.420,179.997,7.619,149.438
C06924=1118.264,72.589,-55.402,179.996,7.615,149.437
C06925=1118.269,72.340,-55.384,179.994,7.611,149.437
C06926=1118.274,72.090,-55.367,179.993,7.606,149.436
C06927=1118.278,71.841,-55.350,179.992,7.603,149.436
C06928=1118.283,71.591,-55.332,179.990,7.599,149.436
C06929=1118.288,71.342,-55.314,179.989,7.596,149.435
C06930=1118.293,71.093,-55.297,179.988,7.591,149.434
C06931=1118.298,70.844,-55.280,179.986,7.587,149.434
C06932=1118.303,70.595,-55.263,179.985,7.583,149.434
C06933=1118.308,70.345,-55.245,179.983,7.579,149.433
C06934=1118.313,70.096,-55.228,179.982,7.575,149.432
C06935=1118.318,69.846,-55.211,179.980,7.571,149.432
C06936=1118.323,69.597,-55.193,179.979,7.567,149.431
C06937=1118.327,69.347,-55.176,179.978,7.563,149.431
C06938=1118.332,69.098,-55.158,179.976,7.559,149.431
C06939=1118.338,68.848,-55.141,179.974,7.555,149.430
C06940=1118.342,68.600,-55.124,179.974,7.552,149.429
C06941=1118.348,68.351,-55.107,179.972,7.548,149.429
C06942=1118.353,68.101,-55.090,179.971,7.544,149.429
C06943=1118.357,67.852,-55.072,179.970,7.540,149.428
C06944=1118.362,67.602,-55.055,179.968,7.536,149.428
C06945=1118.367,67.353,-55.038,179.967,7.532,149.427
C06946=1118.372,67.103,-55.020,179.965,7.528,149.426
C06947=1118.377,66.854,-55.003,179.964,7.524,149.426
C06948=1118.382,66.605,-54.987,179.962,7.520,149.426
C06949=1118.387,66.356,-54.969,179.961,7.516,149.425
C06950=1118.391,66.106,-54.952,179.960,7.512,149.425
C06951=1118.396,65.856,-54.935,179.958,7.508,149.424
C06952=1118.401,65.607,-54.918,179.958,7.504,149.423
C06953=1118.406,65.358,-54.900,179.956,7.500,149.423
C06954=1118.411,65.109,-54.884,179.954,7.496,149.423
C06955=1118.416,64.859,-54.867,179.953,7.492,149.422
C06956=1118.421,64.610,-54.850,179.952,7.488,149.422
C06957=1118.426,64.360,-54.832,179.951,7.484,149.421
C06958=1118.430,64.111,-54.815,179.949,7.480,149.420
C06959=1118.436,63.862,-54.798,179.948,7.476,149.420
C06960=1118.440,63.612,-54.782,179.946,7.472,149.419
C06961=1118.446,63.363,-54.764,179.945,7.468,149.419
C06962=1118.450,63.113,-54.748,179.943,7.464,149.418
C06963=1118.455,62.899,-54.733,179.943,7.461,149.418
C06964=1118.458,62.684,-54.719,179.942,7.457,149.417
C06965=1118.463,62.470,-54.704,179.940,7.453,149.417
C06966=1118.467,62.256,-54.689,179.939,7.450,149.417
C06967=1118.472,62.041,-54.675,179.938,7.447,149.416
C06968=1118.475,61.827,-54.660,179.937,7.443,149.416
C06969=1118.480,61.612,-54.645,179.936,7.440,149.415
C06970=1118.484,61.398,-54.631,179.935,7.437,149.415
C06971=1118.489,61.148,-54.614,179.933,7.433,149.414
C06972=1118.494,60.899,-54.597,179.932,7.429,149.414
C06973=1118.499,60.649,-54.580,179.931,7.425,149.413
C06974=1118.504,60.400,-54.564,179.930,7.421,149.413
C06975=1118.508,60.151,-54.547,179.928,7.417,149.412
C06976=1118.514,59.901,-54.530,179.927,7.413,149.412
C06977=1118.519,59.652,-54.513,179.925,7.409,149.411
C06978=1118.523,59.403,-54.497,179.924,7.405,149.411
C06979=1118.528,59.153,-54.479,179.923,7.400,149.410
C06980=1118.533,58.904,-54.463,179.922,7.397,149.410
C06981=1118.539,58.654,-54.446,179.921,7.393,149.409
C06982=1118.543,58.405,-54.429,179.919,7.389,149.409
C06983=1118.548,58.155,-54.412,179.918,7.385,149.408
C06984=1118.554,57.906,-54.396,179.917,7.381,149.408
C06985=1118.558,57.656,-54.380,179.915,7.377,149.407
C06986=1118.563,57.407,-54.363,179.914,7.373,149.406
C06987=1118.568,57.158,-54.347,179.912,7.369,149.406
C06988=1118.573,56.908,-54.329,179.911,7.364,149.405
C06989=1118.578,56.659,-54.313,179.910,7.361,149.405
C06990=1118.583,56.410,-54.296,179.909,7.357,149.404
C06991=1118.588,56.160,-54.279,179.908,7.353,149.404
C06992=1118.593,55.911,-54.263,179.907,7.349,149.403
C06993=1118.598,55.661,-54.247,179.905,7.345,149.403
C06994=1118.602,55.412,-54.230,179.904,7.341,149.402
C06995=1118.608,55.163,-54.213,179.902,7.337,149.402
C06996=1118.613,54.913,-54.197,179.901,7.332,149.401
C06997=1118.618,54.664,-54.180,179.900,7.328,149.401
C06998=1118.622,54.414,-54.164,179.899,7.324,149.400
C06999=1118.627,54.165,-54.148,179.898,7.321,149.400
C07000=1118.633,53.916,-54.131,179.897,7.317,149.399
C07001=1118.637,53.666,-54.114,179.895,7.313,149.398
C07002=1118.643,53.417,-54.099,179.894,7.309,149.398
C07003=1118.647,53.167,-54.082,179.892,7.305,149.397
C07004=1118.652,52.919,-54.066,179.891,7.300,149.397
C07005=1118.657,52.669,-54.048,179.890,7.296,149.396
C07006=1118.662,52.419,-54.032,179.889,7.292,149.396
C07007=1118.667,52.170,-54.016,179.888,7.288,149.395
C07008=1118.672,51.920,-53.999,179.887,7.285,149.395
C07009=1118.677,51.671,-53.984,179.885,7.280,149.394
C07010=1118.682,51.422,-53.967,179.884,7.276,149.393
C07011=1118.687,51.172,-53.950,179.883,7.272,149.393
C07012=1118.692,50.922,-53.934,179.881,7.268,149.392
C07013=1118.697,50.674,-53.918,179.880,7.264,149.392
C07014=1118.702,50.423,-53.902,179.879,7.260,149.391
C07015=1118.707,50.175,-53.886,179.878,7.256,149.391
C07016=1118.712,49.925,-53.869,179.876,7.251,149.390
C07017=1118.717,49.676,-53.853,179.875,7.248,149.390
C07018=1118.721,49.426,-53.837,179.874,7.244,149.389
C07019=1118.726,49.212,-53.823,179.873,7.240,149.389
C07020=1118.730,48.997,-53.808,179.872,7.237,149.388
C07021=1118.734,48.782,-53.795,179.872,7.233,149.387
C07022=1118.739,48.568,-53.781,179.870,7.230,149.387
C07023=1118.743,48.354,-53.767,179.869,7.226,149.387
C07024=1118.747,48.139,-53.753,179.868,7.223,149.386
C07025=1118.751,47.924,-53.740,179.867,7.219,149.385
C07026=1118.756,47.710,-53.725,179.866,7.216,149.385
C07027=1118.761,47.460,-53.709,179.865,7.212,149.384
C07028=1118.766,47.211,-53.693,179.863,7.208,149.384
C07029=1118.771,46.961,-53.677,179.862,7.203,149.383
C07030=1118.776,46.712,-53.661,179.861,7.199,149.383
C07031=1118.781,46.462,-53.645,179.860,7.195,149.382
C07032=1118.786,46.212,-53.629,179.859,7.191,149.382
C07033=1118.791,45.964,-53.613,179.858,7.187,149.381
C07034=1118.796,45.713,-53.597,179.857,7.183,149.381
C07035=1118.800,45.465,-53.581,179.856,7.179,149.380
C07036=1118.805,45.215,-53.565,179.854,7.175,149.379
C07037=1118.810,44.966,-53.550,179.853,7.171,149.379
C07038=1118.815,44.716,-53.533,179.852,7.167,149.378
C07039=1118.820,44.467,-53.517,179.851,7.162,149.378
C07040=1118.825,44.218,-53.501,179.849,7.158,149.377
C07041=1118.830,43.968,-53.485,179.848,7.154,149.376
C07042=1118.836,43.718,-53.470,179.848,7.151,149.376
C07043=1118.840,43.469,-53.453,179.847,7.146,149.375
C07044=1118.845,43.219,-53.437,179.845,7.142,149.375
C07045=1118.851,42.970,-53.422,179.844,7.138,149.374
C07046=1118.855,42.720,-53.406,179.843,7.134,149.373
C07047=1118.860,42.471,-53.390,179.842,7.129,149.373
C07048=1118.865,42.222,-53.374,179.840,7.125,149.372
C07049=1118.870,41.972,-53.358,179.839,7.121,149.372
C07050=1118.875,41.723,-53.342,179.838,7.117,149.371
C07051=1118.881,41.474,-53.327,179.837,7.113,149.370
C07052=1118.885,41.224,-53.311,179.836,7.109,149.370
C07053=1118.890,40.975,-53.296,179.835,7.105,149.369
C07054=1118.895,40.725,-53.280,179.834,7.101,149.369
C07055=1118.900,40.476,-53.263,179.833,7.097,149.368
C07056=1118.905,40.226,-53.248,179.832,7.092,149.367
C07057=1118.911,39.977,-53.232,179.830,7.088,149.367
C07058=1118.915,39.727,-53.216,179.829,7.084,149.366
C07059=1118.920,39.478,-53.201,179.828,7.080,149.366
C07060=1118.925,39.228,-53.186,179.827,7.075,149.365
C07061=1118.930,38.979,-53.169,179.826,7.071,149.364
C07062=1118.935,38.729,-53.153,179.825,7.068,149.364
C07063=1118.940,38.480,-53.138,179.824,7.064,149.363
C07064=1118.945,38.230,-53.122,179.823,7.059,149.363
C07065=1118.950,37.981,-53.107,179.822,7.055,149.362
C07066=1118.956,37.731,-53.091,179.821,7.051,149.361
C07067=1118.960,37.482,-53.076,179.820,7.046,149.361
C07068=1118.965,37.232,-53.060,179.819,7.042,149.360
C07069=1118.970,36.983,-53.045,179.818,7.038,149.359
C07070=1118.976,36.733,-53.029,179.816,7.034,149.359
C07071=1118.980,36.484,-53.014,179.815,7.030,149.358
C07072=1118.985,36.234,-52.998,179.814,7.025,149.358
C07073=1118.991,35.985,-52.983,179.814,7.022,149.357
C07074=1118.995,35.736,-52.968,179.812,7.017,149.356
C07075=1118.999,35.521,-52.954,179.811,7.013,149.356
C07076=1119.004,35.306,-52.941,179.810,7.010,149.355
C07077=1119.008,35.092,-52.927,179.810,7.006,149.355
C07078=1119.012,34.876,-52.914,179.808,7.003,149.354
C07079=1119.017,34.662,-52.900,179.808,6.999,149.353
C07080=1119.021,34.447,-52.887,179.806,6.995,149.353
C07081=1119.026,34.233,-52.873,179.806,6.992,149.352
C07082=1119.029,34.018,-52.861,179.805,6.988,149.352
C07083=1119.035,33.769,-52.846,179.804,6.984,149.351
C07084=1119.040,33.519,-52.830,179.803,6.980,149.351
C07085=1119.045,33.270,-52.815,179.802,6.975,149.350
C07086=1119.050,33.020,-52.799,179.801,6.971,149.349
C07087=1119.054,32.771,-52.784,179.800,6.967,149.349
C07088=1119.060,32.521,-52.769,179.799,6.963,149.348
C07089=1119.065,32.272,-52.754,179.798,6.958,149.347
C07090=1119.070,32.023,-52.739,179.797,6.954,149.347
C07091=1119.075,31.772,-52.723,179.796,6.950,149.346
C07092=1119.079,31.523,-52.708,179.795,6.945,149.345
C07093=1119.085,31.274,-52.692,179.794,6.942,149.345
C07094=1119.090,31.025,-52.677,179.793,6.937,149.344
C07095=1119.095,30.775,-52.662,179.792,6.933,149.343
C07096=1119.100,30.526,-52.647,179.791,6.929,149.343
C07097=1119.105,30.276,-52.632,179.790,6.925,149.342
C07098=1119.109,30.027,-52.616,179.789,6.920,149.342
C07099=1119.115,29.777,-52.601,179.788,6.916,149.341
C07100=1119.120,29.527,-52.586,179.787,6.911,149.340
C07101=1119.125,29.278,-52.571,179.786,6.907,149.339
C07102=1119.130,29.029,-52.556,179.785,6.903,149.339
C07103=1119.135,28.779,-52.541,179.784,6.898,149.338
C07104=1119.140,28.530,-52.526,179.783,6.894,149.337
C07105=1119.145,28.280,-52.510,179.782,6.890,149.337
C07106=1119.150,28.031,-52.496,179.781,6.885,149.336
C07107=1119.155,27.781,-52.480,179.780,6.882,149.335
C07108=1119.160,27.532,-52.465,179.779,6.877,149.335
C07109=1119.165,27.282,-52.450,179.779,6.873,149.334
C07110=1119.170,27.032,-52.435,179.778,6.868,149.333
C07111=1119.176,26.783,-52.420,179.777,6.864,149.333
C07112=1119.180,26.533,-52.405,179.776,6.860,149.332
C07113=1119.185,26.284,-52.390,179.775,6.856,149.331
C07114=1119.190,26.035,-52.375,179.773,6.851,149.331
C07115=1119.195,25.785,-52.360,179.773,6.846,149.330
C07116=1119.201,25.536,-52.345,179.772,6.842,149.329
C07117=1119.206,25.286,-52.331,179.771,6.838,149.328
C07118=1119.210,25.037,-52.316,179.770,6.834,149.328
C07119=1119.216,24.787,-52.301,179.769,6.829,149.327
C07120=1119.221,24.538,-52.286,179.768,6.825,149.326
C07121=1119.225,24.289,-52.271,179.767,6.820,149.326
C07122=1119.231,24.039,-52.256,179.766,6.816,149.325
C07123=1119.236,23.790,-52.241,179.765,6.812,149.324
C07124=1119.241,23.540,-52.227,179.764,6.807,149.323
C07125=1119.246,23.291,-52.211,179.763,6.803,149.323
C07126=1119.251,23.041,-52.197,179.763,6.799,149.322
C07127=1119.256,22.792,-52.182,179.762,6.795,149.321
C07128=1119.261,22.542,-52.167,179.761,6.790,149.321
C07129=1119.266,22.292,-52.153,179.760,6.786,149.320
C07130=1119.271,22.043,-52.138,179.759,6.781,149.319
C07131=1119.276,21.828,-52.125,179.758,6.777,149.319
C07132=1119.279,21.613,-52.112,179.758,6.774,149.318
C07133=1119.284,21.398,-52.099,179.757,6.769,149.317
C07134=1119.289,21.183,-52.086,179.756,6.766,149.317
C07135=1119.293,20.969,-52.074,179.756,6.762,149.316
C07136=1119.297,20.754,-52.061,179.754,6.758,149.316
C07137=1119.301,20.539,-52.048,179.754,6.755,149.315
C07138=1119.306,20.324,-52.035,179.753,6.750,149.314
C07139=1119.311,20.075,-52.021,179.752,6.746,149.313
C07140=1119.316,19.825,-52.007,179.751,6.741,149.313
C07141=1119.321,19.576,-51.992,179.750,6.737,149.312
C07142=1119.326,19.326,-51.977,179.750,6.732,149.311
C07143=1119.331,19.077,-51.963,179.749,6.728,149.311
C07144=1119.336,18.828,-51.948,179.748,6.724,149.310
C07145=1119.341,18.578,-51.934,179.747,6.719,149.309
C07146=1119.347,18.328,-51.919,179.747,6.715,149.308
C07147=1119.352,18.078,-51.905,179.746,6.711,149.308
C07148=1119.356,17.829,-51.890,179.745,6.706,149.307
C07149=1119.361,17.579,-51.875,179.744,6.702,149.306
C07150=1119.366,17.330,-51.861,179.743,6.697,149.305
C07151=1119.371,17.081,-51.846,179.742,6.693,149.305
C07152=1119.376,16.832,-51.832,179.742,6.688,149.304
C07153=1119.382,16.582,-51.817,179.741,6.684,149.303
C07154=1119.387,16.332,-51.803,179.740,6.679,149.302
C07155=1119.392,16.082,-51.789,179.739,6.675,149.302
C07156=1119.397,15.833,-51.774,179.739,6.670,149.301
C07157=1119.402,15.583,-51.760,179.738,6.666,149.300
C07158=1119.407,15.334,-51.745,179.737,6.661,149.299
C07159=1119.412,15.085,-51.731,179.736,6.657,149.299
C07160=1119.417,14.835,-51.717,179.735,6.652,149.298
C07161=1119.422,14.585,-51.703,179.735,6.648,149.297
C07162=1119.427,14.336,-51.687,179.734,6.643,149.296
C07163=1119.432,14.086,-51.673,179.733,6.638,149.295
C07164=1119.437,13.836,-51.659,179.732,6.634,149.295
C07165=1119.442,13.587,-51.644,179.732,6.629,149.294
C07166=1119.448,13.338,-51.630,179.731,6.625,149.293
C07167=1119.453,13.088,-51.616,179.730,6.620,149.292
C07168=1119.458,12.838,-51.602,179.729,6.615,149.291
C07169=1119.463,12.588,-51.588,179.728,6.611,149.291
C07170=1119.468,12.339,-51.573,179.727,6.606,149.290
C07171=1119.473,12.090,-51.559,179.727,6.601,149.289
C07172=1119.478,11.840,-51.545,179.726,6.597,149.288
C07173=1119.483,11.590,-51.531,179.725,6.592,149.287
C07174=1119.488,11.341,-51.517,179.724,6.588,149.287
C07175=1119.494,11.092,-51.503,179.724,6.583,149.286
C07176=1119.499,10.842,-51.488,179.723,6.578,149.285
C07177=1119.504,10.592,-51.474,179.722,6.574,149.284
C07178=1119.509,10.342,-51.460,179.721,6.569,149.283
C07179=1119.513,10.093,-51.446,179.721,6.565,149.283
C07180=1119.519,9.844,-51.432,179.720,6.560,149.282
C07181=1119.524,9.594,-51.417,179.719,6.556,149.281
C07182=1119.529,9.344,-51.403,179.719,6.551,149.280
C07183=1119.535,9.095,-51.389,179.718,6.546,149.279
C07184=1119.539,8.846,-51.376,179.718,6.541,149.278
C07185=1119.544,8.596,-51.361,179.717,6.537,149.278
C07186=1119.549,8.347,-51.347,179.716,6.532,149.277
C07187=1119.554,8.132,-51.335,179.716,6.529,149.276
C07188=1119.558,7.917,-51.323,179.715,6.524,149.275
C07189=1119.562,7.702,-51.311,179.715,6.521,149.275
C07190=1119.566,7.487,-51.299,179.715,6.517,149.274
C07191=1119.572,7.272,-51.287,179.714,6.512,149.273
C07192=1119.575,7.058,-51.274,179.713,6.509,149.272
C07193=1119.580,6.842,-51.263,179.713,6.505,149.272
C07194=1119.584,6.627,-51.251,179.712,6.501,149.271
C07195=1119.589,6.378,-51.237,179.713,6.497,149.270
C07196=1119.594,6.128,-51.223,179.712,6.492,149.269
C07197=1119.599,5.879,-51.208,179.711,6.488,149.268
C07198=1119.605,5.630,-51.195,179.710,6.483,149.268
C07199=1119.610,5.379,-51.181,179.710,6.478,149.267
C07200=1119.614,5.130,-51.167,179.709,6.473,149.266
C07201=1119.620,4.881,-51.153,179.709,6.470,149.265
C07202=1119.625,4.631,-51.139,179.709,6.465,149.264
C07203=1119.630,4.381,-51.126,179.708,6.460,149.263
C07204=1119.636,4.132,-51.112,179.707,6.456,149.262
C07205=1119.640,3.882,-51.098,179.707,6.451,149.262
C07206=1119.645,3.633,-51.084,179.706,6.446,149.261
C07207=1119.651,3.383,-51.071,179.706,6.442,149.260
C07208=1119.656,3.133,-51.056,179.705,6.438,149.259
C07209=1119.660,2.885,-51.043,179.705,6.433,149.258
C07210=1119.666,2.634,-51.029,179.704,6.429,149.257
C07211=1119.671,2.385,-51.015,179.704,6.424,149.257
C07212=1119.676,2.136,-51.001,179.703,6.419,149.256
C07213=1119.681,1.886,-50.988,179.702,6.415,149.255
C07214=1119.686,1.636,-50.974,179.702,6.410,149.254
C07215=1119.691,1.387,-50.960,179.702,6.406,149.253
C07216=1119.696,1.137,-50.946,179.701,6.402,149.252
C07217=1119.701,0.888,-50.933,179.700,6.397,149.252
C07218=1119.706,0.638,-50.919,179.700,6.392,149.251
C07219=1119.711,0.388,-50.905,179.699,6.388,149.250
C07220=1119.717,0.139,-50.891,179.699,6.383,149.249
C07221=1119.722,-0.111,-50.878,179.698,6.379,149.248
C07222=1119.727,-0.360,-50.865,179.698,6.375,149.247
C07223=1119.732,-0.610,-50.850,179.697,6.370,149.247
C07224=1119.737,-0.859,-50.838,179.697,6.365,149.246
C07225=1119.742,-1.109,-50.823,179.696,6.361,149.245
C07226=1119.747,-1.359,-50.810,179.695,6.356,149.244
C07227=1119.752,-1.608,-50.796,179.695,6.352,149.243
C07228=1119.757,-1.858,-50.783,179.694,6.347,149.243
C07229=1119.762,-2.107,-50.770,179.693,6.342,149.242
C07230=1119.768,-2.357,-50.756,179.693,6.339,149.241
C07231=1119.773,-2.606,-50.742,179.693,6.334,149.240
C07232=1119.778,-2.856,-50.729,179.692,6.330,149.239
C07233=1119.783,-3.105,-50.715,179.691,6.325,149.238
C07234=1119.788,-3.356,-50.702,179.691,6.320,149.237
C07235=1119.793,-3.604,-50.688,179.690,6.316,149.237
C07236=1119.799,-3.855,-50.675,179.689,6.311,149.236
C07237=1119.804,-4.104,-50.662,179.689,6.306,149.235
C07238=1119.809,-4.354,-50.648,179.688,6.302,149.234
C07239=1119.814,-4.603,-50.635,179.687,6.297,149.234
C07240=1119.819,-4.853,-50.621,179.687,6.293,149.233
C07241=1119.825,-5.102,-50.608,179.687,6.289,149.232
C07242=1119.829,-5.352,-50.594,179.686,6.284,149.231
C07243=1119.834,-5.566,-50.583,179.685,6.280,149.230
C07244=1119.838,-5.782,-50.572,179.685,6.276,149.230
C07245=1119.843,-5.997,-50.561,179.684,6.272,149.229
C07246=1119.847,-6.212,-50.549,179.683,6.268,149.228
C07247=1119.851,-6.427,-50.537,179.683,6.265,149.228
C07248=1119.856,-6.642,-50.526,179.683,6.261,149.227
C07249=1119.860,-6.857,-50.514,179.682,6.256,149.226
C07250=1119.865,-7.072,-50.503,179.682,6.253,149.225
C07251=1119.869,-7.321,-50.489,179.681,6.248,149.225
C07252=1119.875,-7.571,-50.476,179.680,6.244,149.224
C07253=1119.879,-7.821,-50.463,179.680,6.239,149.223
C07254=1119.885,-8.070,-50.450,179.679,6.235,149.222
C07255=1119.890,-8.319,-50.437,179.678,6.230,149.221
C07256=1119.895,-8.569,-50.423,179.678,6.225,149.220
C07257=1119.901,-8.819,-50.410,179.677,6.220,149.220
C07258=1119.905,-9.068,-50.396,179.676,6.216,149.219
C07259=1119.911,-9.318,-50.384,179.676,6.211,149.218
C07260=1119.916,-9.568,-50.370,179.675,6.207,149.217
C07261=1119.921,-9.817,-50.357,179.674,6.202,149.216
C07262=1119.926,-10.067,-50.345,179.674,6.198,149.216
C07263=1119.931,-10.316,-50.330,179.674,6.194,149.215
C07264=1119.936,-10.566,-50.318,179.673,6.189,149.214
C07265=1119.941,-10.816,-50.304,179.672,6.185,149.213
C07266=1119.947,-11.065,-50.292,179.672,6.180,149.212
C07267=1119.952,-11.315,-50.279,179.671,6.176,149.212
C07268=1119.957,-11.565,-50.266,179.670,6.171,149.211
C07269=1119.962,-11.814,-50.252,179.670,6.166,149.210
C07270=1119.967,-12.063,-50.240,179.669,6.161,149.209
C07271=1119.972,-12.313,-50.226,179.668,6.157,149.208
C07272=1119.977,-12.563,-50.213,179.668,6.152,149.207
C07273=1119.983,-12.813,-50.200,179.667,6.148,149.206
